// TwinCAT 3 PLC project IBF_Utilities
// Title: IBF_Utilities
// Company: Industrial Brains B.V.
// ProjectVersion: 0.0.0.0
// Description: The utilities library contains all basic utilities needed like system variables, messages, parameters etc.
// ProgramVersion: 3.1.4023.0
// libraries:
//   Tc2_Standard, * (Beckhoff Automation GmbH)
//   Tc2_System, * (Beckhoff Automation GmbH)
//   Tc2_Utilities, * (Beckhoff Automation GmbH)
//   Tc3_EventLogger, * (Beckhoff Automation GmbH)
//   Tc3_Module, * (Beckhoff Automation GmbH)
// project tree:
//   Average/ FB_RollingAverageLREAL.TcPOU (not stored), FB_RollingAverageTime.TcPOU (not stored), F_AverageLREAL.TcPOU (not stored), F_AverageTime.TcPOU (not stored)
//   BaseFunctions/ FB_Base.TcPOU, FB_FunctionBase.TcPOU
//   Compare/Functions/ Between.TcPOU, Between360deg.TcPOU (not stored)
//   Conversion/ DegS_To_Rpm.TcPOU (not stored), DegS_To_Rpm_And_MMin.TcPOU, DT_To_Str.TcPOU, Grey_To_Bin.TcPOU, MMin_To_Rpm_And_DegS.TcPOU (not stored), Rpm_To_DegS.TcPOU
//   FaultsAndMessages/DataTypes/ E_FaultTypes.TcTLEO, E_ResetState.TcDUT, UDT_Fault.TcDUT, UDT_FaultLogItem.TcDUT, UDT_Identity.TcDUT
//   FaultsAndMessages/Functions/ FB_FaultHandler.TcPOU
//   General/DataTypes/ E_ComponentTypes.TcTLEO, E_Locations.TcTLEO, Udt_TimerBandwith.TcDUT
//   GVLs/ DataManager.TcGVL, GVL_FixedValues.TcGVL, GVL_Parameters.TcGVL, GVL_Utilities.TcGVL, PAR_Utilities.TcGVL, Sys_Variables.TcGVL
//   Logger/DataTypes/ UDT_LogHandlerConfig.TcDUT, UDT_LogItem.TcDUT, E_LogLevel.TcDUT
//   Logger/Functions/ FB_Logger.TcPOU
//   Logger/Functions/LogHandlers/DataTypes/ E_LogToDiskState.TcDUT
//   Logger/Functions/LogHandlers/ FB_LogHandlerBase.TcPOU, FB_LogHandler_PersistentArray.TcPOU, FB_LogHandler_ADSLOG.TcPOU, FB_LogHandler_TxtFile.TcPOU
//   MovePathCalculations/ fAccDecCalc.TcPOU (not stored)
//   Parameter/DataTypes/ E_ParameterHandlerState.TcDUT, Udt_Parameter.TcDUT, Udt_ParameterId.TcDUT
//   Parameter/Functions/ FB_ParameterFileHandler.TcPOU, FB_ParameterHandler.TcPOU, F_ParToCsvLine.TcPOU (not stored)
//   PathFunctions/ F_FBNameFromPath.TcPOU (not stored), F_GetLevelFromPath.TcPOU (not stored)
//   / PlcTask.TcTTO
//   Positions/FunctionBlocks/ FB_PositionTrigger.TcPOU (not stored), FB_PositionTrigger_Old.TcPOU (not stored)
//   Positions/Functions/ F_AccDecDistanceFromTime.TcPOU (not stored), F_AccDecDistanceFromVelo.TcPOU (not stored), F_PosCheck.TcPOU, F_TopVelocityFromTime.TcPOU (not stored), F_TriggerPosOffset.TcPOU (not stored)
//   StateMachine/ FB_PauseableStateMachine.TcPOU, FB_StateMachine.TcPOU
//   StepFunctions/ FB_CycleTrigger.TcPOU (not stored), FB_Step.TcPOU
//   System/Functions/DataManagement/ FB_PersistentDataManager.TcPOU
//   System/Functions/ Fb_SystemVariables.TcPOU
//   _TESTS/ FB_Base_Test.TcPOU, PRG_TEST_CONVERSION.TcPOU, PRG_TEST_FB_BASE.TcPOU, PRG_TEST_FB_FAULTHANDLER.TcPOU, PRG_TEST_FB_LOGGER.TcPOU, PRG_TEST_FB_PARAMETERHANDLER.TcPOU, PRG_TEST_FB_PARFILEHANDLER.TcPOU, PRG_TEST_FB_STATEMACHINE.TcPOU, PRG_TEST_FB_PAUSEABLESTATEMACHINE.TcPOU, PRG_TEST_GLOBAL.TcPOU
// real-time tasks:
//   TASK PlcTask: cycle T#10ms, priority 20, ADS port 350

CONFIGURATION IBF_Utilities
    RESOURCE PLC ON TwinCAT3
        TASK PlcTask(INTERVAL := T#10ms, PRIORITY := 20);
        PROGRAM PRG_TEST_GLOBAL WITH PlcTask : PRG_TEST_GLOBAL;
        PROGRAM PRG_TEST_FB_BASE WITH PlcTask : PRG_TEST_FB_BASE;
        PROGRAM PRG_TEST_FB_FAULTHANDLER WITH PlcTask : PRG_TEST_FB_FAULTHANDLER;
        PROGRAM PRG_TEST_FB_PARAMETERHANDLER WITH PlcTask : PRG_TEST_FB_PARAMETERHANDLER;
        PROGRAM PRG_TEST_FB_PARFILEHANDLER WITH PlcTask : PRG_TEST_FB_PARFILEHANDLER;
        PROGRAM PRG_TEST_FB_STATEMACHINE WITH PlcTask : PRG_TEST_FB_STATEMACHINE;
        PROGRAM PRG_TEST_FB_PAUSEABLESTATEMACHINE WITH PlcTask : PRG_TEST_FB_PAUSEABLESTATEMACHINE;
        PROGRAM PRG_TEST_CONVERSION WITH PlcTask : PRG_TEST_CONVERSION;
        PROGRAM PRG_TEST_FB_LOGGER WITH PlcTask : PRG_TEST_FB_LOGGER;
    END_RESOURCE
END_CONFIGURATION

// ---- FaultsAndMessages/DataTypes/E_FaultTypes.TcTLEO
{attribute 'qualified_only'}
{attribute 'to_string'}
TYPE E_FaultTypes : // Fault types, sorted by severity
(
	OM, // Operator message
	OW, // Operator warning
	MC, // Missing condition
	CF, // Cycle Fault
	FF, // Fatal fault
	_ENUM_SIZE // Always the last item in the enumerator
) UINT;
END_TYPE

// ---- FaultsAndMessages/DataTypes/E_ResetState.TcDUT
{attribute 'qualified_only'}
{attribute 'strict'}
TYPE E_ResetState :
(
	Idle,
	ResetFaultTypes,
	WaitForFaults,
	Done
);
END_TYPE

// ---- FaultsAndMessages/DataTypes/UDT_Fault.TcDUT
TYPE UDT_Fault :
STRUCT
	Active 			: BOOL := FALSE;
	FaultType 		: E_FaultTypes;
	Description 	: STRING;
END_STRUCT
END_TYPE

// ---- FaultsAndMessages/DataTypes/UDT_FaultLogItem.TcDUT
TYPE UDT_FaultLogItem :
STRUCT
	bEmpty			: BOOL := TRUE; // This log item is empty (does not contain a fault)
	stFault 		: UDT_Fault;
	Id				: STRING; // Fault ID used for reporting and checking duplicates (not an unique value unless description matches as well)
	StartTime		: DATE_AND_TIME; // Time the fault became active
	EndTime			: DATE_AND_TIME; // Time the fault stopped being active
	nInactiveCycles	: UINT; // The number of PLC cycles the fault hasn't been active 
END_STRUCT
END_TYPE

// ---- FaultsAndMessages/DataTypes/UDT_Identity.TcDUT
TYPE UDT_Identity : // The identity is used for logging and fault handling
STRUCT
	nId				: UINT;
	nParentId		: UDINT; // Id of higher level object if aplicable (0 = no parent)
	nLocationId		: UDINT; // Unique Id calculated from Id and ParentId, used for parameter numbers, and as the parent ID for children
	eComponentType	: E_ComponentTypes;
	sName			: STRING[50];
END_STRUCT
END_TYPE

// ---- General/DataTypes/E_ComponentTypes.TcTLEO
{attribute 'qualified_only'}
{attribute 'strict'}
{attribute 'to_string'}
TYPE E_ComponentTypes :
(
	// No entry
		NA			:= 0,
	// Actuators 
		Cylinder 	:= 10,
		Axis		:= 11,
		Heaters		:= 12,
	// Buttons 
		EstopButton	:= 20,
		EstopBumper	:= 21,	
		Pushbutton 	:= 22,
		Switch		:= 23,
	// I/O
		SafeIO		:= 30,
		Rio_Box		:= 31,
		Rio_Slot	:= 32,
		Encoder		:= 33,
		DiInput		:= 34,
		AnInput		:= 35,
		DiOutput	:= 36,
		AnOutput	:= 37,
	// Drive
		ServoDrive 	:= 40,
	// Operation
		HMI			:= 50,
		RemoteOS	:= 51,
		RemoteDB	:= 52,
	// Assemblies
		Assembly 	:= 60,
		SubAssembly	:= 61,
	// functions
		MainProgram		:= 100,
		StepProgram		:= 101,
		FunctionBlock	:= 102 
)UDINT;
END_TYPE

// ---- General/DataTypes/E_Locations.TcTLEO
{attribute 'qualified_only'}
{attribute 'strict'}
TYPE E_Locations :
(
	MainPLC,
	MainPower_230V, 
	MainPower_24V, 
	MainAirSupply,
	MainScreen,
	MainIO,
	RemoteIO
);
END_TYPE

// ---- General/DataTypes/Udt_TimerBandwith.TcDUT
TYPE Udt_TimerBandwith :
STRUCT
	Minimal	:LREAL;// Timer values, Minimum time
	Nominal	:LREAL;// timer values, nominal time
	Maximum	:LREAL;// Timer values, Maximum time
END_STRUCT
END_TYPE

// ---- Logger/DataTypes/UDT_LogHandlerConfig.TcDUT
TYPE UDT_LogHandlerConfig :
STRUCT
	pLogHandler 		: POINTER TO FB_LogHandlerBase := 0;
	eMinimumLogLevel 	: E_LogLevel := E_LogLevel.TRACE;
END_STRUCT
END_TYPE

// ---- Logger/DataTypes/UDT_LogItem.TcDUT
TYPE UDT_LogItem :
STRUCT
	eLevel 		: E_LogLevel;
	stTimestamp : TIMESTRUCT;
	sMsg 		: STRING[255-2]; // Keep 2 bytes room for CRLF line ending
END_STRUCT
END_TYPE

// ---- Logger/DataTypes/E_LogLevel.TcDUT
{attribute 'qualified_only'}
{attribute 'strict'}
{attribute 'to_string'}
TYPE E_LogLevel : // Log levels, for more info see logger methods DEBUG, INFO, etc
(
	TRACE,
	DEBUG,
	INFO,
	WARN,
	ERROR,
	FATAL
) USINT;
END_TYPE

// ---- Logger/Functions/LogHandlers/DataTypes/E_LogToDiskState.TcDUT
{attribute 'qualified_only'}
{attribute 'strict'}
TYPE E_LogToDiskState : // LogToDisk state
(
	InitializeFBs,
	WaitForCommand,
	OpenOrCreateFile,
	CheckFileSize,
	WriteLogItemPrefix,
	WriteLogItemMessage,
	CloseFile,
	FindObsoleteFiles,
	DeleteFile,
	Error
) UDINT;
END_TYPE

// ---- Parameter/DataTypes/E_ParameterHandlerState.TcDUT
{attribute 'qualified_only'}
{attribute 'strict'}
TYPE E_ParameterHandlerState : // Parameter file handler state
(
	InitializeFBs,
	WaitForCommand,
	OpenExistingFile,
	CreateFile,
	WriteRecord,
	WriteRecordBusy,
	ReadRecord,
	ParseRecord,
	CloseFile,
	Error
);
END_TYPE

// ---- Parameter/DataTypes/Udt_Parameter.TcDUT
TYPE Udt_Parameter :
STRUCT PERSISTENT
	nNumber					: UDINT	 	:= 0						; // [Column 0]Parameter data, parameter number
	sName					: STRING	:= 'No parameter' 			; // [Column 1]Parameter data, Parameter name
	sType					: STRING	:= 'PPar'					; // [Column 2]Parameter data, Type of parameter [Mpar, Cpar, Opar, Ppar]
	sDiscription			: STRING	:= 'No parameter selected'	; // [Column 3]Parameter data, Parmater discription
	fFactory				: LREAL		:= 0						; // [Column 4]Parameter data, Factory standard value
	fMaximum				: LREAL		:= 0						; // [Column 5]Parameter data, Maximum parameter value
	fMinimum				: LREAL		:= 0						; // [Column 6]Parameter data, Minimum parameter value
	sUnit					: STRING	:= 'na'						; // [Column 7]Parameter data, Unit of measurement
	fValue					: LREAL		:= 0						; // [Column 8]Parameter data, Current (active) parameter value
	fSaved					: LREAL		:= 0						; // Parameter data, Saved value or standard setpoint
	fPrepared				: LREAL 	:= 0						; // Parameter data, Prepared value from teach function 
	bTeachable				: BOOL		:= FALSE					; // Teach command for devices 
	bAccepted				: BOOL 		:= FALSE 					; // Parameter value has been accepted
	bLoadedFromPersistent 	: BOOL 									; // The variable has been loaded for persistent memory, Note: No init value.
END_STRUCT
END_TYPE

// ---- Parameter/DataTypes/Udt_ParameterId.TcDUT
TYPE Udt_ParameterId :
STRUCT
	nNumber		: UDINT := 0 	; // parameter number
	sName		: STRING[50] := 'NA' ; // parameter name
	sType		: STRING[4]	:= 'Ppar'	; // parameter type 
	pParameter	: POINTER TO Udt_Parameter ; // pointer to parameter
END_STRUCT
END_TYPE

// ---- GVLs/DataManager.TcGVL
{attribute 'qualified_only'}
VAR_GLOBAL
	FbPersistentManager : FB_PersistentDataManager ;
END_VAR

// ---- GVLs/GVL_FixedValues.TcGVL
{attribute 'qualified_only'}
VAR_GLOBAL CONSTANT
	nINTMAXVALUE	: INT := 32767 		; // Integer maximum value 32767
	nINTMINVALUE	: INT := -32767		; // intiger minimum value -32767
	nDINTMAXVALUE	: DINT:= 2147483647 ; // Double integer maximum value 2,147,483,647
	nDINTMINVALUE	: DINT:= -2147483647; // Double integer minimum value -2,147,483,647
END_VAR

// ---- GVLs/GVL_Parameters.TcGVL
{attribute 'qualified_only'}
VAR_GLOBAL
	fbParameterHandler		: FB_ParameterFileHandler ; // Default parameter handler for visualisation and file handling
	sPARLIST_FILE			: T_MaxString 		:= 'D:\Parameters\ParameterList.csv';(* CSV destination file path and name *)
	sPARLOG_FILE			: T_MaxString 		:= 'D:\Parameters\ParameterLog.csv';(* CSV destination file path and name *)
END_VAR
VAR_GLOBAL CONSTANT
	MAX_PARAMETERS 			: UINT := 1000	;
	PAR_COLUMNS 			: UDINT := 8	;
	MAX_CSV_FIELD_LENGTH	: UDINT := 100	;
	sNetId					: T_AmsNetID		:= '' ;
END_VAR

// ---- GVLs/GVL_Utilities.TcGVL
{attribute 'qualified_only'}
VAR_GLOBAL
	fbFaultHandler : FB_FaultHandler; // The one and only faulthandler (a singleton)
END_VAR
VAR_GLOBAL CONSTANT
	// Not a PAR_Utility, because this constant is used by a HMI list (which is not compatible with configurable constant values)
	RETAINABLE_LOG_HISTORY_SIZE : UINT := 100;
END_VAR

// ---- GVLs/PAR_Utilities.TcGVL
{attribute 'qualified_only'}
// Contains library parameters
VAR_GLOBAL CONSTANT
	MAX_FAULTS_IN_LOG : UINT := 16; // Max number of faults in the FaultHandler log (should match with the size of the HMI's logview table)
END_VAR

// ---- GVLs/Sys_Variables.TcGVL
(* System variables *)
{attribute 'qualified_only'}
VAR_GLOBAL
// SystemFuntion
	fbSystemVariables : Fb_SystemVariables ;
	AlwaysOn		:BOOL 			;// System variable, Always on bit
	AlwaysOff		:BOOL 			;// System variable, Always off bit
	BlinkFast		:BOOL 			;// System variable, Blink fast bit 1sec 
	BlinkSlow		:BOOL 			;// System variable, Blink slow bit 2 sec
	Pulse1Sec		:BOOL 			;// System variable, Pulse 1 cycle every second
	Pulse100ms		:BOOL 			;// System variable, pulse 1 cycle every 100 ms
	SystemTime		:DATE_AND_TIME	; // System variable, Windows system time as DATE_AND_TIME
	SystemTime_TS	:TIMESTRUCT		; // System variable, Windows system time as TIMESTRUCT
	TimeZoneId		:E_TimeZoneID 	; // System variable, time zone Id 
	HeartBeat		:BOOL 			;// System Variable, Main system heartbeat 0.5 sec on 0.5 sec off
END_VAR

// ---- _TESTS/PRG_TEST_GLOBAL.TcPOU
PROGRAM INTERNAL PRG_TEST_GLOBAL // A place to call global function blocks (singletons) that can be used by all tests

Sys_Variables.fbSystemVariables();
GVL_Utilities.fbFaultHandler();

END_PROGRAM

// ---- _TESTS/PRG_TEST_FB_BASE.TcPOU
PROGRAM INTERNAL PRG_TEST_FB_BASE
VAR
	bEnableTests : BOOL;
	fbBase : FB_Base_Test;
END_VAR

IF bEnableTests THEN
	fbBase.Init(1, 2, E_ComponentTypes.MainProgram);
	fbBase();
END_IF

END_PROGRAM

// ---- _TESTS/FB_Base_Test.TcPOU
FUNCTION_BLOCK INTERNAL FB_Base_Test EXTENDS FB_Base

SUPER^();

METHOD PUBLIC Init : BOOL
VAR_INPUT
	nId				: UINT ; // Identification number of object
	nParentId		: UINT ; // Id of higher level if applicable (0 = no parent)
	eComponentType	: E_ComponentTypes ; // Component or function type
END_VAR
// Every FB_Base instance is expected to have an Init method that calls ExecIdentifyDevice. 
// This Init method will have at least the nId and nParentId inputs.
// The eComponentType input is optional (can be hardcoded in the Init method, for example see FB_Step).
// It might also have additional inputs (changing the method signature) therefore it is not declared in FB_Base.
ExecIdentifyDevice(nId,	nParentId,	eComponentType);
END_METHOD

END_FUNCTION_BLOCK

// ---- BaseFunctions/FB_Base.TcPOU
{attribute 'reflection'}
FUNCTION_BLOCK PUBLIC ABSTRACT FB_Base
VAR_INPUT
	bEnable			: BOOL 		:= TRUE 	; // Module enable signal reference Default := TRUE (when using system library := GVL_Main.stModules[nModuleId].bEnabled)
	refFbParHandler	: REFERENCE TO FB_ParameterFileHandler := GVL_Parameters.fbParameterHandler	; // reference to parameter handler
	bCmdPause 		: BOOL 		:= FALSE	; // Command Pause functions		
END_VAR
VAR_OUTPUT
	stIdentity 		: UDT_Identity;
	bInitOk			: BOOL 			:= FALSE 	; // function is initialized
	bBusy 			: BOOL 			:= FALSE 	; // device is busy
	bReady			: BOOL 			:= FALSE 	; // device is ready for new command 
	bErrorActive	: BOOL			:= FALSE	; // device Error active 
END_VAR
VAR
	stFault			: UDT_Fault		; // Fault data from device

	// Function path 
	{attribute 'instance-path'} 
    {attribute 'noinit'}
	sPath			: STRING	; // Path name of function (used for manual reference)
END_VAR

GVL_Utilities.fbFaultHandler.CmdAddFault(
	stFault := stFault,
	stIdentity := stIdentity
);

METHOD PUBLIC CmdReset : BOOL
VAR_INPUT
END_VAR
bErrorActive := FALSE ;

CmdReset := TRUE ;
END_METHOD

METHOD PROTECTED ExecIdentifyDevice : BOOL
VAR_INPUT
	nId				: UINT; // Identification number of object (between 0 and 99)
	nParentId		: UDINT; // Id of higher level If aplicable (0 = no parent)
	eComponentType	: E_ComponentTypes; // Component or function type
END_VAR
stIdentity.nId := nId;
stIdentity.nParentId := nParentId;
stIdentity.eComponentType := eComponentType;
stIdentity.sName := F_FBNameFromPath(sPath := sPath);
stIdentity.nLocationId := stIdentity.nParentId * 10000 + stIdentity.nId * 100;

ExecIdentifyDevice := (stIdentity.sName <> '') AND (stIdentity.nId < 100);
END_METHOD

END_FUNCTION_BLOCK

// ---- Parameter/Functions/FB_ParameterFileHandler.TcPOU
FUNCTION_BLOCK FB_ParameterFileHandler EXTENDS FB_ParameterHandler
VAR CONSTANT
	sCSVFileHeader 	: STRING := 'NUMBER;NAME;TYPE;DESCRIPTION;FACTORY;MAXIMUM;MINIMUM;UNIT;VALUE$L';
	CSV_FIELDS 		: UINT := 9;
END_VAR
VAR_OUTPUT
	bFault : BOOL;
	sFaultDescription : STRING;
END_VAR
VAR
	// States
	eState 		: E_ParameterHandlerState := E_ParameterHandlerState.InitializeFBs;
	
	// Command helpers
	bDone 		: BOOL;
	bCmdInit 	: BOOL;
	bCmdSavePar : BOOL;
	
	// File function blocks (asynchronous)
	fbFileOpen	: FB_FileOpen; // https://infosys.beckhoff.com/content/1033/tcplclib_tc2_system/30977547.html
	fbFileWrite	: FB_FileWrite; // https://infosys.beckhoff.com/content/1033/tcplclib_tc2_system/30986763.html
	fbFileClose	: FB_FileClose; // https://infosys.beckhoff.com/content/1033/tcplclib_tc2_system/30972939.html
	fbFileGets	: FB_FileGets; // https://infosys.beckhoff.com/content/1033/tcplclib_tc2_system/30976011.html

	// CSV handling
	sCsvRecord : T_MaxString := ''; // String buffer (single CSV text line)
	bHeaderRead : BOOL; // TRUE once the CSV header line has been read
	fbCsvMemBufReader : FB_CSVMemBufferReader; // https://infosys.beckhoff.com/content/1033/tcplclib_tc2_utilities/34977931.html
	fbCsvMemBufWriter : FB_CSVMemBufferWriter; // https://infosys.beckhoff.com/content/1033/tcplclib_tc2_utilities/34979467.html

	// Miscelleanous
	nIdxPar  : UINT; // Parameter array iterator
END_VAR

ExecStateMachine();

METHOD PUBLIC CmdSavePar : BOOL
IF NOT bCmdSavePar THEN
	bDone := FALSE;
	bCmdSavePar := TRUE;
ELSIF bDone THEN
	bCmdSavePar := FALSE;
END_IF	

CmdSavePar := bDone;
END_METHOD

METHOD PRIVATE ExecStateMachine : BOOL
VAR
	i 					: UINT; // Iterator
	pParameter 			: POINTER TO Udt_Parameter; // Temporary pointer to parameter
	sParameterFromFile 	: Udt_Parameter; // Parameter retrieved from file
	sCSVField 			: T_MaxString; // Single CSV field value (record field)
	bMatch 				: BOOL;
END_VAR
// Parameter file handler state machine
CASE eState OF
	E_ParameterHandlerState.InitializeFBs:
		// Initialize function blocks
		fbFileOpen(
			bExecute := FALSE,
			ePath := PATH_GENERIC,
		);
		fbFileWrite(
			bExecute := FALSE,
			pWriteBuff := ADR(sCsvRecord)
		);
		fbFileClose(bExecute := FALSE);
		fbFileGets(bExecute := FALSE);

		fbCsvMemBufWriter.pBuffer := ADR(sCsvRecord);
		fbCsvMemBufReader.pBuffer := ADR(sCsvRecord);
		fbCsvMemBufWriter.cbBuffer := SIZEOF(sCsvRecord) - 1;
		fbCsvMemBufReader.cbBuffer := SIZEOF(sCsvRecord);
	
		eState := E_ParameterHandlerState.WaitForCommand;

	E_ParameterHandlerState.WaitForCommand:
		sFaultDescription := '';
		IF bCmdInit THEN
			eState := E_ParameterHandlerState.OpenExistingFile;
		ELSIF bCmdSavePar THEN
			eState := E_ParameterHandlerState.CreateFile;
		END_IF	

	E_ParameterHandlerState.OpenExistingFile:
		fbFileOpen(
			bExecute := TRUE,	
			sPathName := GVL_Parameters.sPARLIST_FILE,
			nMode := FOPEN_MODEREAD OR FOPEN_MODETEXT, // Open file in read only text mode
		);

		IF (NOT fbFileOpen.bBusy) THEN
			fbFileOpen(bExecute := FALSE);

			IF fbFileOpen.bError THEN
				// Check error codes
				IF (fbFileOpen.nErrId = 16#70C) THEN
					// File not found
					eState := E_ParameterHandlerState.CreateFile;
				ELSE
					sFaultDescription := 'Unable to open file';
					eState := E_ParameterHandlerState.Error;
				END_IF
			ELSE
				nIdxPar := 0;
				bHeaderRead := FALSE;
				eState := E_ParameterHandlerState.ReadRecord;
			END_IF
		END_IF

	E_ParameterHandlerState.CreateFile:
		fbFileOpen(
			bExecute := TRUE,	
			sPathName := GVL_Parameters.sPARLIST_FILE,
			nMode := FOPEN_MODEWRITE OR FOPEN_MODETEXT, // Open file in read/write text mode
		);

		IF (NOT fbFileOpen.bBusy) THEN
			fbFileOpen(bExecute := FALSE);

			IF fbFileOpen.bError THEN
				sFaultDescription := 'Unable to create file';
				eState := E_ParameterHandlerState.Error;
			ELSE		
				fbFileWrite.hFile := fbFileOpen.hFile;
				nIdxPar := 0;
				eState := E_ParameterHandlerState.WriteRecord;
			END_IF
		END_IF
		
	E_ParameterHandlerState.WriteRecord:
		// Code based on Beckhoff example: https://infosys.beckhoff.com/content/1033/tcplclib_tc2_utilities/34979467.html
		sCsvRecord := '';
		fbCsvMemBufWriter.eCmd := eEnumCmd_First; // Write first field value

		IF (nIdxPar > nNumberOfParameters) THEN
			// Done (all parameters were added)
			eState := E_ParameterHandlerState.CloseFile;
		ELSIF (nIdxPar = 0) THEN
			// First line: write the CSV header
			sCsvRecord := sCSVFileHeader;
			eState := E_ParameterHandlerState.WriteRecordBusy;
		ELSE
			// Add the next parameter
			pParameter := arParameters[nIdxPar].pParameter;
			IF (pParameter = 0) THEN
				sFaultDescription := 'Unexpected null pointer';
				eState := E_ParameterHandlerState.Error;
			ELSE
				// Save current actual value for later restore
				pParameter^.fSaved := pParameter^.fValue;
				// Create CSV record
				FOR i := 1 TO CSV_FIELDS DO 
					CASE i OF
						1: sCSVField := UDINT_TO_STRING(pParameter^.nNumber);
						2: sCSVField := pParameter^.sName;
						3: sCSVField := pParameter^.sType;
						4: sCSVField := pParameter^.sDiscription;
						5: sCSVField := LREAL_TO_STRING(pParameter^.fFactory);
						6: sCSVField := LREAL_TO_STRING(pParameter^.fMaximum);
						7: sCSVField := LREAL_TO_STRING(pParameter^.fMinimum);
						8: sCSVField := pParameter^.sUnit;
						9: sCSVField := LREAL_TO_STRING(pParameter^.fValue);
					END_CASE
					sCSVField := STRING_TO_CSVFIELD(sCSVField, FALSE);
					
					// Add new field to the record buffer
					fbCsvMemBufWriter(
						putValue := sCSVField,
						bCRLF := (i = CSV_FIELDS) // Write CRLF after the last field value 
					);
					IF fbCsvMemBufWriter.bOk THEN
						fbCsvMemBufWriter.eCmd := eEnumCmd_Next;
					ELSE // Error
						sFaultDescription := 'Unable to store fields in CSV buffer';
						eState := E_ParameterHandlerState.Error;
						RETURN;
					END_IF
	
				END_FOR

				eState := E_ParameterHandlerState.WriteRecordBusy;
			END_IF;
		END_IF;

	E_ParameterHandlerState.WriteRecordBusy:
		fbFileWrite(bExecute := TRUE, cbWriteLen := INT_TO_UDINT(LEN(sCsvRecord)));
		IF (NOT fbFileWrite.bBusy) THEN
			fbFileWrite(bExecute := FALSE);
			IF fbFileWrite.bError THEN
				sFaultDescription := 'Unable to write record to file';
				eState := E_ParameterHandlerState.Error;
			ELSE		
				nIdxPar := nIdxPar + 1;	 
				eState := E_ParameterHandlerState.WriteRecord;
			END_IF
		END_IF
		
	E_ParameterHandlerState.ReadRecord:
		fbFileGets(bExecute := TRUE, hFile := fbFileOpen.hFile);
		IF (NOT fbFileGets.bBusy) THEN
			sCsvRecord := fbFileGets.sLine;
			fbFileGets(bExecute := FALSE);
			IF fbFileGets.bError THEN
				sFaultDescription := 'Unable to read line from file';
				eState := E_ParameterHandlerState.Error;
			ELSIF fbFileGets.bEOF THEN
				// Finished reading the file
				eState := E_ParameterHandlerState.CloseFile;			
			ELSIF NOT bHeaderRead THEN 
				// Skip first line (header)
				bHeaderRead := TRUE;
			ELSE
				eState := E_ParameterHandlerState.ParseRecord;
			END_IF
		END_IF

	E_ParameterHandlerState.ParseRecord:
		fbCsvMemBufReader.eCmd := eEnumCmd_First; // Read first field value

		FOR i := 1 TO CSV_FIELDS DO 
			// Read field from the record buffer
			fbCsvMemBufReader(getValue => sCSVField);
			IF fbCsvMemBufReader.bOk THEN
				sCSVField := CSVFIELD_TO_STRING(sCSVField, FALSE);
				CASE i OF
					1: sParameterFromFile.nNumber := STRING_TO_UDINT(sCSVField);
					2: sParameterFromFile.sName := sCSVField;
					3: sParameterFromFile.sType := sCSVField;
					4: sParameterFromFile.sDiscription := sCSVField;
					5: sParameterFromFile.fFactory := STRING_TO_LREAL(sCSVField);
					6: sParameterFromFile.fMaximum := STRING_TO_LREAL(sCSVField);
					7: sParameterFromFile.fMinimum := STRING_TO_LREAL(sCSVField);
					8: sParameterFromFile.sUnit := sCSVField;
					9: sParameterFromFile.fValue := STRING_TO_LREAL(sCSVField);
				END_CASE
				
				fbCsvMemBufReader.eCmd := eEnumCmd_Next;
			ELSE // Error
				sFaultDescription := 'Unable to parse all CSV fields';
				eState := E_ParameterHandlerState.Error;
				RETURN;
			END_IF
		END_FOR
			
		// Done reading parameter from file. Search for parameter in the PLC parameter array, and copy values.
		FOR i := 1 TO nNumberOfParameters DO
			pParameter := arParameters[i].pParameter;
			IF (pParameter = 0) THEN
				// Unexpected null pointer
				EXIT;
			ELSIF (sParameterFromFile.nNumber = pParameter^.nNumber) THEN
				bMatch := TRUE;
				pParameter^.sName := sParameterFromFile.sName;
				pParameter^.sType := sParameterFromFile.sType;
				pParameter^.sDiscription := sParameterFromFile.sDiscription;
				pParameter^.fFactory := sParameterFromFile.fFactory;
				pParameter^.fMaximum := sParameterFromFile.fMaximum;
				pParameter^.fMinimum := sParameterFromFile.fMinimum;
				pParameter^.sUnit := sParameterFromFile.sUnit;
				pParameter^.fValue := sParameterFromFile.fValue;
				EXIT;
			END_IF
		END_FOR

		IF bMatch THEN
			// Finished, move to the next record		
			eState := E_ParameterHandlerState.ReadRecord;
		ELSE
			sFaultDescription := 'Parameter in CSV file not found in PLC';
			eState := E_ParameterHandlerState.Error;
		END_IF
	
	E_ParameterHandlerState.CloseFile:
		fbFileClose(bExecute := TRUE, hFile := fbFileOpen.hFile);
		IF (NOT fbFileClose.bBusy) THEN
			fbFileClose(bExecute := FALSE);
			IF fbFileClose.bError THEN
				sFaultDescription := 'Unable to close file'; 
				eState := E_ParameterHandlerState.Error;
			ELSE
				bDone := TRUE;
				eState := E_ParameterHandlerState.WaitForCommand;
			END_IF
		END_IF
	
	E_ParameterHandlerState.Error:
		IF (sFaultDescription = '') THEN
			sFaultDescription := 'Unknown error';
		END_IF

END_CASE

bFault := (eState = E_ParameterHandlerState.Error);
END_METHOD

METHOD PUBLIC Init : BOOL
IF NOT bCmdInit THEN
	bDone := FALSE;
	bCmdInit := TRUE;
ELSIF bDone THEN
	bCmdInit := FALSE;
END_IF	

Init := bDone;
END_METHOD

END_FUNCTION_BLOCK

// ---- Parameter/Functions/FB_ParameterHandler.TcPOU
FUNCTION_BLOCK PUBLIC FB_ParameterHandler
VAR_OUTPUT
	arParameters		: ARRAY [1..GVL_Parameters.MAX_PARAMETERS] OF Udt_ParameterId := [stDummyParId]; 
END_VAR
VAR
	nLookupIndex		: UINT := 1;
	nNumberOfParameters : UINT := 1;
	// parameter change commands
	bCmdLoadfactory		: BOOL 	:= FALSE; // Load factory value into prepared value 
	bCmdLoadFromPrevious: BOOL 	:= FALSE; // Load from saved previous value into prepared value
	bCmdTeach			: BOOL 	:= FALSE; // Start teaching function for selected parameter
	bCmdAcceptTeach		: BOOL 	:= FALSE ; // Accept the teach value
	// Dummy parameter when no parameters are added yet
	stDummyParId		: Udt_ParameterId ;
	// Memory 
	fValueOld			: LREAL	:= 0 ; // previous value
END_VAR

// call parameter change function 
ExecChangeParValues();

METHOD PUBLIC CmdAddParameter : BOOL
VAR_IN_OUT
	refParameter : Udt_Parameter ; // Parameter to add
END_VAR
VAR
	i 			: UINT ;
	j			: UINT ;
	stTempPar	: Udt_ParameterId ;
	bParFound	: BOOL 	:= FALSE ;
END_VAR
//Single loop to get the number of parameters and check if that parameter has already been added  
FOR i := 1 TO GVL_Parameters.MAX_PARAMETERS DO
	//Check if it's a valid reference
	IF (arParameters[i].pParameter = 0) THEN
		//No, we have reached the end of the list
		//The current index - 1 is the ammount of parameters
		nNumberOfParameters := i - 1;
		//Abort the FOR loop, we found the end.
		EXIT ;
	//It is a valid reference, valitate it is not already in the list  
	ELSIF arParameters[i].nNumber = refParameter.nNumber THEN
		//It is in the list, validate if the name matches 
		IF (arParameters[i].sName = refParameter.sName) THEN
			//Name and number match, assume it is the same parameter and just return that it is (already) added
			CmdAddParameter := TRUE;
			RETURN;
		ELSE
			//Number matches but not the name, this is a different parameter. Abort the add.
			CmdAddParameter := FALSE;
			RETURN;
		END_IF
	END_IF
END_FOR

//Ok, here we are shure it's a new parameter, try adding it to the array
nNumberOfParameters := nNumberOfParameters + 1; 
//Does it fit?
IF nNumberOfParameters <= GVL_Parameters.MAX_PARAMETERS THEN
	//It fits, store the data
	arParameters[nNumberOfParameters].nNumber		:= refParameter.nNumber 	;
	arParameters[nNumberOfParameters].sName			:= refParameter.sName	;
	arParameters[nNumberOfParameters].sType			:= refParameter.sType	;
	arParameters[nNumberOfParameters].pParameter 	:= ADR(refParameter)	;
	
	//Check if the add was sucessfull
	CmdAddParameter := arParameters[nNumberOfParameters].pParameter <> 0;
	
	//Give the command to (re)sort the parameter list
	ExecSortParameters();
ELSE
	//Does not fit, return FALSE
	CmdAddParameter := FALSE;	
END_IF
END_METHOD

METHOD ExecChangeParValues : BOOL
VAR
END_VAR
IF arParameters[nLookupIndex].pParameter <> 0 THEN 
	;
ELSE
	RETURN; 
END_IF

// Load values from default or saved
IF bCmdLoadfactory THEN 
	arParameters[nLookupIndex].pParameter^.fValue := arParameters[nLookupIndex].pParameter^.fFactory ;
	bCmdLoadfactory := FALSE ;
ELSIF bCmdLoadFromPrevious THEN
	arParameters[nLookupIndex].pParameter^.fValue := arParameters[nLookupIndex].pParameter^.fSaved ;
	bCmdLoadFromPrevious := FALSE ;
ELSIF bCmdAcceptTeach THEN 
	arParameters[nLookupIndex].pParameter^.fValue := arParameters[nLookupIndex].pParameter^.fPrepared ;
	bCmdAcceptTeach := FALSE ;
END_IF
END_METHOD

METHOD PRIVATE ExecSortParameters : BOOL
VAR_INPUT
END_VAR
VAR
	i 			: UDINT ;
	j			: UDINT ;
	stTempPar	: Udt_ParameterId ;
END_VAR
// (re)sort parameter list so it's order remains constant
FOR i := 2 TO nNumberOfParameters BY 1 DO
	FOR j := 1 TO nNumberOfParameters - 1 BY 1 DO
		IF (arParameters[j].nNumber > arParameters[j+1].nNumber)THEN
			stTempPar 			:= arParameters[j+1];
			arParameters[j+1]	:= arParameters[j];
			arParameters[j]		:= stTempPar ;
		END_IF
	END_FOR
END_FOR
END_METHOD

END_FUNCTION_BLOCK

// ---- _TESTS/PRG_TEST_FB_FAULTHANDLER.TcPOU
PROGRAM INTERNAL PRG_TEST_FB_FAULTHANDLER
VAR
	bEnableTests : BOOL;
	fbBase : FB_Base_Test;
	bCmdReset : BOOL;
	bCmdClearInactive : BOOL;
	stLogItem : UDT_FaultLogItem;
	bHead : BOOL;
	bNext : BOOL;
	bActive : BOOL;
	pFault : POINTER TO UDT_Fault; // Workaround to reach non-output variable fbBase.stFault
END_VAR

IF bEnableTests THEN
	fbBase();
	
	pFault := ADR(fbBase.stFault);
	pFault^.Active := bActive;
	
	IF bCmdReset THEN
		bCmdReset R= GVL_Utilities.fbFaultHandler.CmdReset();
	END_IF
	
	IF bCmdClearInactive THEN
		bCmdClearInactive R= GVL_Utilities.fbFaultHandler.CmdClearInactive();
	END_IF
	
	IF bHead THEN
		bHead := FALSE;
		stLogItem := GVL_Utilities.fbFaultHandler.Head;
	END_IF

	IF bNext THEN
		bNext := FALSE;
		stLogItem := GVL_Utilities.fbFaultHandler.Next;
	END_IF
END_IF

END_PROGRAM

// ---- _TESTS/PRG_TEST_FB_PARAMETERHANDLER.TcPOU
PROGRAM INTERNAL PRG_TEST_FB_PARAMETERHANDLER
VAR
	bEnableTests : BOOL;
	fbParameterHandler 	: FB_ParameterHandler;
	stParameterId		: Udt_ParameterId;
	stParameter 		: Udt_Parameter; // NOTE: Udt_Parameter is persistent
	bAddParameter 		: BOOL;
END_VAR

IF bEnableTests THEN
	fbParameterHandler();
	
	IF bAddParameter THEN
		bAddParameter := FALSE;
		fbParameterHandler.CmdAddParameter(stParameter);
	END_IF
END_IF

END_PROGRAM

// ---- _TESTS/PRG_TEST_FB_PARFILEHANDLER.TcPOU
PROGRAM INTERNAL PRG_TEST_FB_PARFILEHANDLER
VAR
	bEnableTests : BOOL;
	fbParFileHandler: FB_ParameterFileHandler;
	stParameter 	: Udt_Parameter; // NOTE: Udt_Parameter is persistent
	bAddParameter 	: BOOL;
	bInit			: BOOL;
	bCmdSavePar		: BOOL;
END_VAR

IF bEnableTests THEN
	fbParFileHandler();
	
	IF bAddParameter THEN
		bAddParameter := FALSE;
		fbParFileHandler.CmdAddParameter(stParameter);
	END_IF
	
	IF bInit THEN
		bInit R= fbParFileHandler.Init();
	END_IF
	
	IF bCmdSavePar THEN
		bCmdSavePar R= fbParFileHandler.CmdSavePar();
	END_IF
END_IF

END_PROGRAM

// ---- _TESTS/PRG_TEST_FB_STATEMACHINE.TcPOU
PROGRAM INTERNAL PRG_TEST_FB_STATEMACHINE
VAR
	bEnableTests : BOOL;
	nState : UDINT;
	fbStateMachine : FB_StateMachine;
	bStateChanged : BOOL; // A helper variable to detect bStateChanged output changes in FB_StateMachine
	nTimeInState : UDINT; // [msec] A helper variable to get the elapsed time as a number 
END_VAR

IF bEnableTests THEN
	fbStateMachine(nState := nState);
	bStateChanged S= fbStateMachine.bStateChanged;
	nTimeInState := TIME_TO_UDINT(fbStateMachine.tTimeInState);
END_IF

END_PROGRAM

// ---- StateMachine/FB_StateMachine.TcPOU
FUNCTION_BLOCK FB_StateMachine // A basic statemachine with some convenient outputs
VAR CONSTANT
	MAX_TIME : TIME := UDINT_TO_TIME(16#FFFFFFFF);
END_VAR
VAR_IN_OUT
	nState : UDINT;
END_VAR
VAR_OUTPUT
	tTimeInState : TIME;
	bStateChanged : BOOL;
END_VAR
VAR
	nStatePrev : UDINT;
	tonTimeInState : TON;
END_VAR

bStateChanged := (nStatePrev <> nState);
nStatePrev := nState;
tonTimeInState(IN := NOT bStateChanged, PT := MAX_TIME);
tTimeInState := tonTimeInState.ET;

END_FUNCTION_BLOCK

// ---- _TESTS/PRG_TEST_FB_PAUSEABLESTATEMACHINE.TcPOU
PROGRAM INTERNAL PRG_TEST_FB_PAUSEABLESTATEMACHINE
VAR CONSTANT
	PAUSE_STATE : UDINT := 100;
END_VAR
VAR
	bEnableTests : BOOL;

	nState : UDINT;
	fbStateMachine : FB_PauseableStateMachine;
	bDoSomething : BOOL;
END_VAR

IF bEnableTests THEN
	fbStateMachine(nState := nState, nPauseState := PAUSE_STATE);
	
	CASE nState OF
		0 : IF bDoSomething THEN
				nState := 1;
			END_IF
			
		PAUSE_STATE :
			IF bDoSomething THEN
				 fbStateMachine.Resume();
			END_IF
	END_CASE

	bDoSomething := FALSE;
END_IF

END_PROGRAM

// ---- StateMachine/FB_PauseableStateMachine.TcPOU
FUNCTION_BLOCK FB_PauseableStateMachine EXTENDS FB_StateMachine // An extension of FB_StateMachine that allows state pauses
VAR_INPUT
	nPauseState : UDINT; // The state to go to when paused
	bRequestPause : BOOL; // If TRUE, the state machine will go to nPauseState on the next state change
	bIgnorePause : BOOL; // If TRUE, the state machine will ignore a pause request. NOTE: This BOOL will be set to FALSE on a state change
END_VAR
VAR
	nResumeState : UDINT; // The state to go to when un-pausing (where the statemachine wanted to go, but wasn' allowed to) 
END_VAR

SUPER^(nState := nState);

IF bStateChanged THEN
	IF bRequestPause AND (NOT bIgnorePause) THEN
		nResumeState := nState;
		nState := nPauseState;
		nStatePrev := nState;
	END_IF
	bIgnorePause := FALSE;
END_IF

METHOD PUBLIC Resume
{warning disable C0371}
IF __ISVALIDREF(nState) THEN
	IF (NOT bRequestPause) THEN
		nState := nResumeState;
	END_IF
END_IF
{warning restore C0371}
END_METHOD

END_FUNCTION_BLOCK

// ---- _TESTS/PRG_TEST_CONVERSION.TcPOU
PROGRAM INTERNAL PRG_TEST_CONVERSION
VAR
 	bEnableTests : BOOL;

	in_dt : DATE_AND_TIME;
	out_str : STRING;
END_VAR

IF bEnableTests THEN
	out_str := Dt_To_Str(in_dt);
END_IF

END_PROGRAM

// ---- Conversion/DT_To_Str.TcPOU
FUNCTION DT_To_Str : STRING[19] // Takes a DATE_AND_TIME and converts it into a atring. If 0, an empty string is returned 
VAR_INPUT
	value : DATE_AND_TIME;
END_VAR
VAR
	str : STRING;
END_VAR

IF (DT_TO_DWORD(value) = 0) THEN
	DT_To_Str := '';
ELSE
	// Example input: 'DT#1998-02-13-14:20:00
	str := MID(DT_TO_STRING(value), 19, 4); // Cut off 'DT#'
	str := REPLACE(str, ' ', 1, 11); // Take out unnecessary '-'
	DT_To_Str :=  str;
END_IF

END_FUNCTION

// ---- _TESTS/PRG_TEST_FB_LOGGER.TcPOU
PROGRAM INTERNAL PRG_TEST_FB_LOGGER
VAR
	fbLogHandler_TxtFile :	FB_LogHandler_TxtFile(
									sLogFolder := 'D:\Temp\',
									sLogFilePrefix := 'AutomaticTestLog_',
									sLogFileExtension := 'txt',
									nMaxLogFileSize := 500,
									nMaxNumberOfLogFiles := 3
								);
	fbLogHandler_ADSLOG : FB_LogHandler_ADSLOG;
	fbLogger : FB_Logger;
	
	bRegisterLogHandlers : BOOL;
	bEnableTests : BOOL;
	bAddToLog : BOOL;
	eLogLevel : E_LogLevel;
	bStressTest : BOOL;
	nIdx : UDINT;
	sMsg : T_MaxString;
END_VAR

IF bEnableTests THEN
	IF bRegisterLogHandlers THEN
		fbLogger.RegisterLogHandler(fbLogHandler_ADSLOG, E_LogLevel.TRACE);
		fbLogger.RegisterLogHandler(fbLogHandler_TxtFile, E_LogLevel.TRACE);
	END_IF
	
	fbLogger.Run();
	
	IF bAddToLog THEN
		bAddToLog := FALSE;
		CASE eLogLevel OF
			E_LogLevel.TRACE:	fbLogger.TRACE(sMsg);
			E_LogLevel.DEBUG: 	fbLogger.DEBUG(sMsg);
			E_LogLevel.INFO: 	fbLogger.INFO(sMsg);
			E_LogLevel.WARN: 	fbLogger.WARN(sMsg);
			E_LogLevel.ERROR:	fbLogger.ERROR(sMsg);
			E_LogLevel.FATAL: 	fbLogger.FATAL(sMsg);
		END_CASE
	END_IF
	
	IF bStressTest THEN
		// Write an item to the log every PLC cycle, this should trigger a buffer overflow
		nIdx := nIdx + 1;
		sMsg := UDINT_TO_STRING(nIdx);
		fbLogger.TRACE(sMsg);
	END_IF
END_IF

END_PROGRAM

// ---- Logger/Functions/LogHandlers/FB_LogHandler_TxtFile.TcPOU
FUNCTION_BLOCK PUBLIC FB_LogHandler_TxtFile EXTENDS FB_LogHandlerBase // Regularly writes contents of the log to disk
// Once the log file reaches a set size, a new log file is created.
// If the max number of files is reached, the oldest file is discarded.
VAR CONSTANT
	MAX_ITEMS_IN_BUFFER : UDINT := 20; // Should be long enough to allow for worst case writes (where an old file has to be deleted and a new file created).  
END_VAR
VAR_OUTPUT
	bFault 				: BOOL; // An error occured while trying to add to log or write to disk
	sFaultDescription	: STRING[80]; // Detailed error information
	bLoggerInitialized  : BOOL; // True the first time the logger has ran through all states (ie., after succesfully writing the first log message and emptying the buffer)
	sCurrentLogFile		: T_MaxString; // The file which is currently used for logging (and can be viewed for instance by the HMI)
END_VAR
VAR
	// Properties set by FB_init
	sLogFolder 			: T_MaxString;
	sLogFilePrefix 		: T_MaxString;
	sLogFileExtension 	: T_MaxString;
	nMaxLogFileSize 	: ULINT; // [bytes] When this size is reached, a new log file is created 
	nMaxNumberOfLogFiles: UINT;

	// State machine
	fbStateMachine 	: FB_StateMachine;	
	eState 			: E_LogToDiskState := E_LogToDiskState.InitializeFBs;
	
	// Log item buffer
	stLogItemFromBuffer : UDT_LogItem; // Log item retrieved from the buffer	
	stLogItemToDisk		: UDT_LogItem; // Log item to be written to the log file
	cbBuffer 	: ARRAY[1..(MAX_ITEMS_IN_BUFFER * (SIZEOF(UDT_LogItem) + 4))] OF BYTE; // Note that the buffer size is larger than the number of items * item size, because 4 bytes are added to each item by FB_MemRingBuffer
	fbBuffer 	: FB_MemRingBuffer := (pBuffer:= ADR(cbBuffer), cbBuffer:= SIZEOF(cbBuffer));

	// File function blocks (asynchronous)
	fbFileOpen			: FB_FileOpen; // https://infosys.beckhoff.com/content/1033/tcplclib_tc2_system/30977547.html
	fbFilePuts			: FB_FilePuts; // https://infosys.beckhoff.com/content/1033/tcplclib_tc2_system/30979083.html
	fbFileClose			: FB_FileClose; // https://infosys.beckhoff.com/content/1033/tcplclib_tc2_system/30972939.html
	fbFileProperties	: FB_FileProperties; // https://infosys.beckhoff.com/content/1033/tcplclib_tc2_utilities/10047843595.html
    fbEnumFiles			: FB_EnumFindFileEntry; // https://infosys.beckhoff.com/content/1033/tcplclib_tc2_utilities/34982539.html
	fbFileDelete		: FB_FileDelete; // https://infosys.beckhoff.com/content/1033/tcplclib_tc2_system/30974475.html

	sPath: STRING; // Path to the current log file
	
	tOldestLogFile 	: ST_FindFileEntry; // Reference to the oldest log file in the log folder
	nFileCount		: UINT; // Number of log files found  
	
	fbFormatString : FB_FormatString; // https://infosys.beckhoff.com/content/1033/tcplclib_tc2_utilities/34990219.html
END_VAR
VAR_TEMP
	sTimestamp : T_MaxString;
	sLevel : T_MaxString;

	nFileSize : ULINT;
	
	stEmptyLogItem : UDT_LogItem;
END_VAR

fbStateMachine(nState := eState);

CASE eState OF
	E_LogToDiskState.InitializeFBs:
		// Initialize function blocks
		fbFileOpen(
			bExecute := FALSE,
			ePath := PATH_GENERIC,
		);
		fbFilePuts(bExecute := FALSE);
		fbFileClose(bExecute := FALSE);
		fbFileProperties(bExecute := FALSE);
		fbEnumFiles(bExecute := FALSE);
		fbFileDelete(
			bExecute := FALSE,
			ePath := PATH_GENERIC,
		);
		
		eState := E_LogToDiskState.WaitForCommand;

	E_LogToDiskState.WaitForCommand:
		IF (stLogItemFromBuffer.sMsg = '') THEN
			stLogItemFromBuffer := Pop();
		ELSE
			eState := E_LogToDiskState.OpenOrCreateFile;
		END_IF

	E_LogToDiskState.OpenOrCreateFile:
		IF fbStateMachine.bStateChanged THEN
			// Create a new file path if none was given (i.e., after reboot or when file size limit has been reached)
			IF (sPath = '') THEN
				sPath := CreatePath();
			END_IF  	
		END_IF
		fbFileOpen(
			bExecute := TRUE,	
			sPathName := sPath, 
			nMode := FOPEN_MODEAPPEND OR FOPEN_MODETEXT, // Open file in read/write text mode
		);
		IF (NOT fbFileOpen.bBusy) THEN
			fbFileOpen(bExecute := FALSE);
			IF fbFileOpen.bError THEN
				fbFormatString(sFormat := 'Unable to open file (error code 0x%X)', arg1 := F_UDINT(fbFileOpen.nErrId), sOut => sFaultDescription);
				eState := E_LogToDiskState.Error;
			ELSE
				sCurrentLogFile := sPath;
				eState := E_LogToDiskState.CheckFileSize;
			END_IF
		END_IF

	E_LogToDiskState.CheckFileSize:
		fbFileProperties(
			bExecute := TRUE,	
			sPathName := sPath 
		);
		IF (NOT fbFileProperties.bBusy) THEN
			fbFileProperties(bExecute := FALSE);
			IF fbFileProperties.bError THEN
				fbFormatString(sFormat := 'Unable to get file properties (error code 0x%X)', arg1 := F_UDINT(fbFileProperties.nErrId), sOut => sFaultDescription);
				eState := E_LogToDiskState.Error;
			ELSE
				// Check file size
				// ST_FindFileEntry info at https://infosys.beckhoff.com/content/1033/tcplclib_tc2_utilities/35363851.html
				nFileSize := ULARGE_TO_ULINT(fbFileProperties.stProperties.fileSize);
				IF (nFileSize >= nMaxLogFileSize) THEN
					// Create a final log item for this log file
					stLogItemToDisk.eLevel := E_LogLevel.DEBUG;
					fbFormatString(
						sFormat := 'File size exceeded (%u/%u bytes), creating new file.',
						arg1 := F_ULINT(nFileSize),
						arg2 := F_ULINT(nMaxLogFileSize),
						sOut => stLogItemToDisk.sMsg
					);
					stLogItemToDisk.stTimestamp := Sys_Variables.SystemTime_TS;
					sPath := ''; // Trigger new file creation
				ELSE
					stLogItemToDisk := stLogItemFromBuffer; // Set log item to be written to disk
					stLogItemFromBuffer := stEmptyLogItem; // Clear log item from buffer to trigger new item pop
				END_IF
				eState := E_LogToDiskState.WriteLogItemPrefix;
			END_IF
		END_IF
	
	E_LogToDiskState.WriteLogItemPrefix:
		IF fbStateMachine.bStateChanged THEN
			// Build a prefix string, e.g. '[2022-02-04 12:13:45.343] INFO; '

			// Suppress error "VAR_IN_OUT parameter 'in' needs variable with write access as input."	
			sLevel := TO_STRING(stLogItemToDisk.eLevel);
			sTimestamp := SYSTEMTIME_TO_STRING(stLogItemToDisk.stTimestamp);
 
			fbFormatString(
				sFormat := '[%s] %s: ',
				arg1 := F_STRING(sTimestamp),
				arg2 := F_STRING(sLevel),
				sOut => fbFilePuts.sLine
			);
		END_IF
		fbFilePuts(bExecute := TRUE, hFile := fbFileOpen.hFile);
		IF (NOT fbFilePuts.bBusy) THEN
			fbFilePuts(bExecute := FALSE);
			IF fbFilePuts.bError THEN
				fbFormatString(sFormat := 'Unable to write log record to file (error code 0x%X)', arg1 := F_UDINT(fbFilePuts.nErrId), sOut => sFaultDescription);
				eState := E_LogToDiskState.Error;
			ELSE // Done, write the log message
				eState := E_LogToDiskState.WriteLogItemMessage;
			END_IF
		END_IF
	
	E_LogToDiskState.WriteLogItemMessage:
		IF fbStateMachine.bStateChanged THEN
			fbFilePuts.sLine := CONCAT(stLogItemToDisk.sMsg, '$L'); // Add line feed character
		END_IF
		fbFilePuts(bExecute := TRUE, hFile := fbFileOpen.hFile);
		IF (NOT fbFilePuts.bBusy) THEN
			fbFilePuts(bExecute := FALSE);
			IF fbFilePuts.bError THEN
				fbFormatString(sFormat := 'Unable to write log record to file (error code 0x%X)', arg1 := F_UDINT(fbFilePuts.nErrId), sOut => sFaultDescription);
				eState := E_LogToDiskState.Error;
			ELSE // Done, get the next log item in the buffer
				IF (stLogItemFromBuffer.sMsg <> '') THEN 
					// Last log item retrieved from the buffer wasn't written yet (e.g., after new file creation), so no need to pop items from the buffer yet
					eState := E_LogToDiskState.CloseFile;
				ELSE // Check if there are more items in the buffer
					stLogItemFromBuffer := Pop();
					IF (stLogItemFromBuffer.sMsg = '') THEN // Buffer empty, close the file
						eState := E_LogToDiskState.CloseFile;
					ELSE // More items to be written, but first check file size before adding more items
						eState := E_LogToDiskState.CheckFileSize;
					END_IF
				END_IF
			END_IF
		END_IF
	
	E_LogToDiskState.CloseFile:
		fbFileClose(bExecute := TRUE, hFile := fbFileOpen.hFile);
		IF (NOT fbFileClose.bBusy) THEN
			fbFileClose(bExecute := FALSE);
			IF fbFileClose.bError THEN
				fbFormatString(sFormat := 'Unable to close file (error code 0x%X)', arg1 := F_UDINT(fbFileClose.nErrId), sOut => sFaultDescription);
				eState := E_LogToDiskState.Error;
			ELSE
				eState := E_LogToDiskState.FindObsoleteFiles;
			END_IF
		END_IF
	
	E_LogToDiskState.FindObsoleteFiles:
		// Delete oldest log files in log folder until we're at MAX_NUMBER_OF_LOG_FILES
		IF fbStateMachine.bStateChanged THEN
			nFileCount := 0;	
			tOldestLogFile.sFileName := ''; 
			// Create a path search string, e.g. '/tmp/Log_*.txt'
			fbFormatString(
				sFormat := '%s%s*.%s',
				arg1 := F_STRING(sLogFolder),
				arg2 := F_STRING(sLogFilePrefix),
				arg3 := F_STRING(sLogFileExtension),
				sOut => fbEnumFiles.sPathName
			);
			fbEnumFiles.eCmd := E_EnumCmdType.eEnumCmd_First;
		END_IF
		fbEnumFiles(bExecute := TRUE);
		IF (NOT fbEnumFiles.bBusy) THEN
			fbEnumFiles(bExecute := FALSE, eCmd := E_EnumCmdType.eEnumCmd_Next);
			IF fbEnumFiles.bError THEN
				fbFormatString(
					sFormat := 'Unable to get files in folder "%s" (error code 0x%X)',
					arg1 := F_STRING(fbEnumFiles.sPathName),
					arg2 := F_UDINT(fbEnumFiles.nErrId),
					sOut => sFaultDescription
				);
				eState := E_LogToDiskState.Error;
			ELSIF fbEnumFiles.bEOE THEN
				// Found all files, carry on
				eState := E_LogToDiskState.WaitForCommand;
				bLoggerInitialized := TRUE;
			ELSE
				// Found a file, check if it's older than the previous find
				nFileCount := nFileCount + 1;
				IF (tOldestLogFile.sFileName = '') 
					OR (PLWORD_TO_LWORD(ADR(fbEnumFiles.stFindFile.creationTime)) < PLWORD_TO_LWORD(ADR(tOldestLogFile.creationTime))) 
				THEN
					tOldestLogFile := fbEnumFiles.stFindFile;
				END_IF
				IF (nFileCount > nMaxNumberOfLogFiles) THEN
					// Max number of log files reached, delete the file				
					eState := E_LogToDiskState.DeleteFile;
				END_IF
			END_IF
		END_IF

	E_LogToDiskState.DeleteFile:
		IF fbStateMachine.bStateChanged THEN
			fbFormatString(
				sFormat := '%s%s',
				arg1 := F_STRING(sLogFolder),
				arg2 := F_STRING(tOldestLogFile.sFileName),
				sOut => fbFileDelete.sPathName
			);
		END_IF
		fbFileDelete(bExecute := TRUE);
		IF (NOT fbFileDelete.bBusy) THEN
			fbFileDelete(bExecute := FALSE);
			IF fbFileDelete.bError THEN
				fbFormatString(
					sFormat := 'Unable to delete file "%s" (error code 0x%X)',
					arg1 := F_STRING(tOldestLogFile.sFileName),
					arg2 := F_UDINT(fbFileClose.nErrId), 
					sOut => sFaultDescription
				);
				eState := E_LogToDiskState.Error;
			ELSE // Done deleting, continue searching for obsolete files
				eState := E_LogToDiskState.FindObsoleteFiles;
			END_IF
		END_IF

	E_LogToDiskState.Error:
		IF (sFaultDescription = '') THEN
			sFaultDescription := 'Unknown error';
		END_IF

END_CASE

bFault S= (eState = E_LogToDiskState.Error);

METHOD INTERNAL FINAL AddToLog
VAR_INPUT
	stLogItem : UDT_LogItem;
END_VAR
VAR
	bOk : BOOL;
	nMaxItems : UDINT;
END_VAR
// Ignore incoming items when the logger has an error
IF bFault THEN
	RETURN;
END_IF


fbBuffer.A_AddTail(
	pWrite := ADR(stLogItem),
	cbWrite := SIZEOF(stLogItem),
	bOk => bOk,
);

IF NOT bOk THEN // Buffer overflow
	// Make sure no more items will be added to the log
	bFault := TRUE;
	// Pop last item to make room for the famous last words
	Pop(); 
	// And add those words to the log
	nMaxItems := MAX_ITEMS_IN_BUFFER;
	fbFormatString(
		sFormat := 'Log buffer size limit (%u) reached! Dumping buffer and disabling the log handler.',
		arg1 := F_UDINT(nMaxItems),
		sOut => sFaultDescription
	);
	stLogItem.sMsg := sFaultDescription;
	stLogItem.eLevel := E_LogLevel.FATAL;
	fbBuffer.A_AddTail(
		pWrite := ADR(stLogItem),
		cbWrite := SIZEOF(stLogItem),
		bOk => bOk,
	);
END_IF
END_METHOD

METHOD PROTECTED CreatePath : STRING // Create a filename with a date/time stamp, e.g. "/tmp/Log_20230203-093610.txt'
VAR
	fMonth : REAL;
	fDay : REAL;
	fHour : REAL;
	fMinute : REAL;
	fSecond : REAL;
END_VAR
// Suppress error "VAR_IN_OUT parameter 'in' needs variable with write access as input."	
fMonth := WORD_TO_REAL(Sys_Variables.SystemTime_TS.wMonth); 
fDay := WORD_TO_REAL(Sys_Variables.SystemTime_TS.wDay); 
fHour := WORD_TO_REAL(Sys_Variables.SystemTime_TS.wHour); 
fMinute := WORD_TO_REAL(Sys_Variables.SystemTime_TS.wMinute); 
fSecond := WORD_TO_REAL(Sys_Variables.SystemTime_TS.wSecond); 

fbFormatString(
	sFormat := '%s%s%u%02.0f%02.0f-%02.0f%02.0f%02.0f.%s',
	arg1 := F_STRING(sLogFolder),
	arg2 := F_STRING(sLogFilePrefix),
	arg3 := F_WORD(Sys_Variables.SystemTime_TS.wYear),
	arg4 := F_REAL(fMonth),
	arg5 := F_REAL(fDay),
	arg6 := F_REAL(fHour),
	arg7 := F_REAL(fMinute),
	arg8 := F_REAL(fSecond),
	arg9 := F_STRING(sLogFileExtension),
	sOut => CreatePath
);
END_METHOD

METHOD FB_init : BOOL
VAR_INPUT
	bInitRetains : BOOL; // if TRUE, the retain variables are initialized (warm start / cold start)
	bInCopyCode : BOOL;  // if TRUE, the instance afterwards gets moved into the copy code (online change)

	sLogFolder 			: T_MaxString; // Example for TwinCAT/BSD: '/tmp/'. The folder where log files will be stored. Add trailing '/' or '\'. 
	sLogFilePrefix 		: T_MaxString; // Example: 'Log_'
	sLogFileExtension 	: T_MaxString; // Example: 'txt'
	nMaxLogFileSize 	: ULINT; // [bytes] When this size is reached, a new log file is created 
	nMaxNumberOfLogFiles: UINT;
END_VAR
THIS^.sLogFolder := sLogFolder;
IF (sLogFolder = '') THEN
	bFault := TRUE;
	sFaultDescription := 'Parameter "sLogFolder" empty';
END_IF
THIS^.sLogFilePrefix := sLogFilePrefix;
THIS^.sLogFileExtension := sLogFileExtension;
THIS^.nMaxLogFileSize := nMaxLogFileSize;
THIS^.nMaxNumberOfLogFiles := nMaxNumberOfLogFiles;
END_METHOD

METHOD PROTECTED Pop : UDT_LogItem; // Pops the buffer head (returns the oldest log item in the buffer)
fbBuffer.A_RemoveHead(
	pRead:= ADR(Pop),
	cbRead:= SIZEOF(Pop),
);
END_METHOD

END_FUNCTION_BLOCK

// ---- Logger/Functions/LogHandlers/FB_LogHandlerBase.TcPOU
{attribute 'reflection'}
FUNCTION_BLOCK PUBLIC ABSTRACT FB_LogHandlerBase // Base class for all log handlers
VAR_OUTPUT
	{attribute 'instance-path'} 
    {attribute 'noinit'}
	sInstancePath : STRING; // Instance path of the function block
END_VAR

METHOD INTERNAL ABSTRACT AddToLog
VAR_INPUT
	stLogItem : UDT_LogItem;
END_VAR
END_METHOD

END_FUNCTION_BLOCK

// ---- Logger/Functions/LogHandlers/FB_LogHandler_ADSLOG.TcPOU
FUNCTION_BLOCK FB_LogHandler_ADSLOG EXTENDS FB_LogHandlerBase // Writes log item to the ADS log
VAR
END_VAR

METHOD INTERNAL FINAL AddToLog
VAR_INPUT
	stLogItem : UDT_LogItem;
END_VAR
VAR
	msgCtrlMask : DWORD; // ADS log message control mask, more info: https://infosys.beckhoff.com/content/1033/tcplclib_tc2_system/31030539.html	
END_VAR
msgCtrlMask := ADSLOG_MSGTYPE_LOG OR ADSLOG_MSGTYPE_STRING;
CASE stLogItem.eLevel OF
	E_LogLevel.TRACE: 	msgCtrlMask := msgCtrlMask OR ADSLOG_MSGTYPE_HINT;
	E_LogLevel.DEBUG: 	msgCtrlMask := msgCtrlMask OR ADSLOG_MSGTYPE_HINT;
	E_LogLevel.INFO: 	msgCtrlMask := msgCtrlMask OR ADSLOG_MSGTYPE_HINT;
	E_LogLevel.WARN: 	msgCtrlMask := msgCtrlMask OR ADSLOG_MSGTYPE_WARN;
	E_LogLevel.ERROR:	msgCtrlMask := msgCtrlMask OR ADSLOG_MSGTYPE_ERROR;
	E_LogLevel.FATAL: 	msgCtrlMask := msgCtrlMask OR ADSLOG_MSGTYPE_ERROR;
END_CASE

ADSLOGSTR(
	msgCtrlMask := msgCtrlMask,
	msgFmtStr := '%s',
	strArg := stLogItem.sMsg
);
END_METHOD

END_FUNCTION_BLOCK

// ---- Logger/Functions/FB_Logger.TcPOU
FUNCTION_BLOCK PUBLIC FB_Logger
VAR_STAT
	aLogHandlers : ARRAY[1..10] OF UDT_LogHandlerConfig; // The log handlers that process the incoming log messages
	bUnexpectedCall : BOOL; // FB_Logger should never be called. Use this bit to avoid flooding the log.
END_VAR

IF NOT bUnexpectedCall THEN
	THIS^.FATAL('Unexpected call to FB_Logger(). Do not call FB_Logger!');
	bUnexpectedCall := TRUE;
END_IF

METHOD PUBLIC DEBUG // Add a message to the log with log level DEBUG 
(*
The DEBUG level is used for logging messages that help developers find out what went wrong
during a debugging session. While the specifics of what messages to log at the DEBUG level
is dependent on your application, you generally want to include detailed information that
can help developers troubleshoot an issue quickly. 
This can include variable state in the surrounding scope, or relevant error codes.
Unlike TRACE, DEBUG level logging can be turned on in production without making the application unusable,
but it should not be left on indefinitely to ensure the log is not flooded.
*)
VAR_INPUT
	sMsg : T_MaxString; // The message to be logged
END_VAR
THIS^.SendToLogHandlers(sMsg, E_LogLevel.DEBUG);
END_METHOD

METHOD PUBLIC ERROR // Add a message to the log with log level ERROR
(*
The ERROR log level is used to represent error conditions in a system that
prevent a specific operation from running, but the system itself can continue
working even if it is at a reduced level of functionality or performance.
Generally, ERROR logs should be investigated as soon as possible but they don't
carry the same urgency as FATAL messages since the system can continue working.
*)
VAR_INPUT
	sMsg : T_MaxString; // The message to be logged
END_VAR
THIS^.SendToLogHandlers(sMsg, E_LogLevel.ERROR);
END_METHOD

METHOD PUBLIC FATAL // Add a message to the log with log level FATAL
(*
The FATAL log level annotates messages with the greatest severity.
It usually means that something critical is broken, and the system cannot continue to do any more
useful work without the intervention of an engineer. T
ypically, such entries are logged before the system is shut down ("famous last words").
*)
VAR_INPUT
	sMsg : T_MaxString; // The message to be logged
END_VAR
THIS^.SendToLogHandlers(sMsg, E_LogLevel.FATAL);
END_METHOD

METHOD PUBLIC INFO // Add a message to the log with log level INFO
(*
INFO-level messages indicate events in the system that are significant to the
general purpose of the system. Such events are logged to show that the system is
operating normally. For example, a recipe was started or stopped. 
Production systems typically default to logging at this level so that a 
summary of the application's normal behavior is visible to anyone reading the logs.
*)
VAR_INPUT
	sMsg : T_MaxString; // The message to be logged
END_VAR
THIS^.SendToLogHandlers(sMsg, E_LogLevel.INFO);
END_METHOD

METHOD PUBLIC RegisterLogHandler : BOOL
VAR_IN_OUT
	fbLogHandler : FB_LogHandlerBase;
END_VAR
VAR_INPUT
	eMinimumLogLevel : E_LogLevel;
END_VAR
VAR
	i : USINT; // Iterator
END_VAR
RegisterLogHandler := TRUE;
FOR i := 1 TO 10 DO
	IF aLogHandlers[i].pLogHandler = ADR(fbLogHandler) THEN // Already added
		RETURN;
	ELSIF aLogHandlers[i].pLogHandler = 0 THEN // Found empty spot in the array, add the log handler
		aLogHandlers[i].pLogHandler := ADR(fbLogHandler);
		aLogHandlers[i].eMinimumLogLevel := eMinimumLogLevel;
		RegisterLogHandler := TRUE;
		DEBUG(CONCAT('Added log handler: ', fbLogHandler.sInstancePath));
		RETURN;
	END_IF
END_FOR
RegisterLogHandler := FALSE; // Failed to add loghandler
END_METHOD

METHOD PUBLIC Run // Enables the logger and log handlers, should be called once every PLC cycle in your program/project (not multiple calls per cycle!)
VAR
	i : USINT; // Iterator
END_VAR
// Call every log handler. Only relevant for log handlers that take multiple PLC cycles
// to handle incoming log items (e.g., writing log items to disk).
FOR i := 1 TO 10 DO
	IF aLogHandlers[i].pLogHandler <> 0 THEN
		aLogHandlers[i].pLogHandler^();
	END_IF
END_FOR
END_METHOD

METHOD PRIVATE SendToLogHandlers
VAR_INPUT
	sMsg : T_MaxString; // The message to be logged
	eLevel : E_LogLevel; // Log level (debug, info, warn, etc.)
END_VAR
VAR
	stLogItem : UDT_LogItem;
	i : USINT; // Iterator
END_VAR
// Ignore empty messages
IF (sMsg = '') THEN
	RETURN;
END_IF

// Create a log item
stLogItem.sMsg := sMsg;
stLogItem.eLevel := eLevel;
stLogItem.stTimestamp := Sys_Variables.SystemTime_TS;

// Add item to all registered loghandlers (if level is high enough)
FOR i := 1 TO 10 DO
	IF (aLogHandlers[i].pLogHandler <> 0) AND (eLevel >= aLogHandlers[i].eMinimumLogLevel) THEN
		aLogHandlers[i].pLogHandler^.AddToLog(stLogItem);
	END_IF
END_FOR
END_METHOD

METHOD PUBLIC TRACE // Add a message to the log with log level TRACE
(*
The TRACE level can be used for tracing the path of code execution in a program.
Generally, TRACE is used for showing the flow of the program, and to provide a detailed breakdown of the sequence
of events that led to a crash, a silent failure, an error, or some other event logged at a different level.
The TRACE level is only used temporarily (when the code is a "work in progress").
*)
VAR_INPUT
	sMsg : T_MaxString; // The message to be logged
END_VAR
THIS^.SendToLogHandlers(sMsg, E_LogLevel.TRACE);
END_METHOD

METHOD PUBLIC WARN // Add a message to the log with log level WARN
(*
Messages logged at the WARN level typically indicate that something unexpected happened,
but the system can recover and continue to function normally.
It is mainly used to draw attention to situations that should be addressed soon before
they pose a problem for the system.
*)
VAR_INPUT
	sMsg : T_MaxString; // The message to be logged
END_VAR
THIS^.SendToLogHandlers(sMsg, E_LogLevel.WARN);
END_METHOD

END_FUNCTION_BLOCK

// ---- System/Functions/DataManagement/FB_PersistentDataManager.TcPOU
FUNCTION_BLOCK FB_PersistentDataManager
VAR_INPUT
END_VAR
VAR_OUTPUT
END_VAR
VAR
	FbWritePersistentData : FB_WritePersistentData ;
	cmdWrite : BOOL := FALSE ;
	TOfWriteInterval	: TOf ;
	CmdWriteFromTime	: BOOL ; 
	TestjeWritten		: BOOL ;
END_VAR

// ===== persistent write interval =====
 TOfWriteInterval(	IN := cmdWrite OR NOT TOfWriteInterval.Q,
	 				PT	:= T#5M  );

IF NOT TOfWriteInterval.Q THEN 
	cmdWrite := TRUE ;
END_IF

// ===== write persistent data =====
	FbWritePersistentData ( PORT 	:= 851,
							START 	:= CmdWrite,
							TMOUT 	:= T#1S,	
							mode 	:= E_PersistentMode.SPDM_VAR_BOOST );	

IF cmdWrite AND FbWritePersistentData.BUSY THEN 
	cmdWrite := FALSE ;
END_IF

METHOD PUBLIC Write : BOOL
VAR_INPUT
END_VAR
IF NOT FbWritePersistentData.BUSY THEN 
	cmdWrite := TRUE ;
ELSE 
	Write := TRUE ;
END_IF
END_METHOD

END_FUNCTION_BLOCK

// ---- FaultsAndMessages/Functions/FB_FaultHandler.TcPOU
FUNCTION_BLOCK FB_FaultHandler
(* 
The faulthandler is responsible for 
	- providing the means for objects to register their faults
	- reporting the active fault types (i.e., message, fatal fault, etc.) --> arActiveFaultTypes
	- providing the means to reset a fault type
	- keeping a log of all faults

It is not responsible for
	- resetting the actual fault (this is up to the object that registered the fault)
	- handling any HMI related functionality

Active faults do not disappear from the log, the need to be manually cleared by issuing a CmdReset and CmdClearInactive.
*)
VAR_INPUT
	nMaxInactiveCycles : UINT := 50; // Once faults haven't been activated for a number of PLC cycles, deactivate them. 0 = do not automatically deactivate faults 
END_VAR
VAR_OUTPUT
	arFaultLog 			: ARRAY [1..PAR_Utilities.MAX_FAULTS_IN_LOG] OF UDT_FaultLogItem;
	nFaultsInLog 		: UINT;
	nActiveFaults 		: UINT;
	arActiveFaultTypes 	: ARRAY[0..(E_FaultTypes._ENUM_SIZE - 1)] OF BOOL; // Status of each fault type
END_VAR
VAR
	fbLogger : FB_Logger;

	bCmdReset : BOOL;
	eResetState : E_ResetState;
	arActiveFaultTypes_Internal : ARRAY[0..(E_FaultTypes._ENUM_SIZE - 1)] OF BOOL; // The actual status of each fault type, which is reported unless the reset cycle is active
	
	nLogIndex : UINT; // Array index of the last added item in the log (zero until the first item arrives)
	nIterIndex : UINT; // Index of the fault log iterator (used for properties First and Next)

	fbFormatString : FB_FormatString; // https://infosys.beckhoff.com/content/1033/tcplclib_tc2_utilities/34990219.html
END_VAR

UpdateInactiveCycles();

ExecReset();

UpdateActiveFaultStatus();

METHOD PROTECTED AddFaultToLog
VAR_INPUT
	stFaultLogItem : UDT_FaultLogItem;
	bActivated : BOOL; // TRUE means the fault has just been activated, FALSE means it stopped being active
END_VAR
VAR
	sStatus : T_MaxString;
	sFaultType : T_MaxString;
	sId : T_MaxString;
	sDescription : T_MaxString;
	sMsg : T_MaxString;
END_VAR
IF bActivated THEN
	sStatus := 'START';
ELSE
	sStatus := 'END';
END_IF
sFaultType := TO_STRING(stFaultLogItem.stFault.FaultType);
sId := stFaultLogItem.Id;
sDescription := stFaultLogItem.stFault.Description;

fbFormatString(
	sFormat := '[%s %s] %s - %s',
	arg1 := F_STRING(sFaultType),
	arg2 := F_STRING(sStatus),
	arg3 := F_STRING(sId),
	arg4 := F_STRING(sDescription),
	sOut => sMsg
);

CASE stFaultLogItem.stFault.FaultType OF
	E_FaultTypes.OM: fbLogger.INFO(sMsg); 
	E_FaultTypes.OW: fbLogger.WARN(sMsg); 
	E_FaultTypes.MC: fbLogger.WARN(sMsg); 
	E_FaultTypes.CF: fbLogger.WARN(sMsg); 
	E_FaultTypes.FF: fbLogger.ERROR(sMsg); 
END_CASE
END_METHOD

METHOD PUBLIC CmdAddFault : BOOL
(*
CmdAddFault should be called every cycle.
If the fault is active, it's corresponding fault type is enabled.
Updates the fault log.
*)
VAR_IN_OUT
	stFault : UDT_Fault; // active fault structure input
END_VAR
VAR_INPUT
	stIdentity : UDT_Identity;
END_VAR
// Update the log
UpdateLog(stFault, stIdentity);

// Clear active status (to be updated by caller)
stFault.Active := FALSE;
END_METHOD

METHOD PUBLIC CmdClearInactive : BOOL // Remove inactive faults from the log
VAR
	stEmptyItem : UDT_FaultLogItem;
	i : UINT; // Iterator
END_VAR
nFaultsInLog := PAR_Utilities.MAX_FAULTS_IN_LOG;
IF (eResetState = E_ResetState.Idle) THEN
	FOR i := 1 TO PAR_Utilities.MAX_FAULTS_IN_LOG DO
		IF (NOT arFaultLog[i].stFault.Active) THEN
			nFaultsInLog :=nFaultsInLog - 1;
			arFaultLog[i] := stEmptyItem;
			arFaultLog[i].bEmpty := TRUE;
		END_IF
	END_FOR
	CmdClearInactive := TRUE;
ELSE
	CmdClearInactive := FALSE;
END_IF
END_METHOD

METHOD PUBLIC CmdReset : BOOL // Reset faults; caller is responsible for stopping the call once TRUE is returned
VAR_INPUT
END_VAR
// Trigger the reset cycle
IF (eResetState = E_ResetState.Idle) THEN
	bCmdReset := TRUE;
END_IF

CmdReset := (eResetState = E_ResetState.Done); // Let the caller know when the reset cycle is finished
END_METHOD

METHOD PRIVATE ExecReset : BOOL
VAR
	i : UINT; // Iterator
END_VAR
CASE eResetState OF
	E_ResetState.Idle: // Wait for reset command
		IF bCmdReset THEN
			// Start the reset cycle
			bCmdReset := FALSE;
			eResetState := E_ResetState.ResetFaultTypes;
		ELSE
			ReportActiveFaultStatus();
		END_IF
	E_ResetState.ResetFaultTypes: 
		// During a reset, the active fault types are not updated 
		// This avoids that faults are not reported for 1 PLC cycle, even though they are still active
		// We do however clear the internal fault types, which are updated automatically during the WaitForFaults state.
		FOR i:= 0 TO (E_FaultTypes._ENUM_SIZE - 1) DO		
			arActiveFaultTypes_Internal[i] := FALSE;
		END_FOR
		eResetState := E_ResetState.WaitForFaults;

	E_ResetState.WaitForFaults: // Allow the PLC one cycle to re-add faults
		eResetState := E_ResetState.Done;

	E_ResetState.Done: // Done, report & allow caller one cycle to reset itself
		ReportActiveFaultStatus();
		eResetState := E_ResetState.Idle;
END_CASE
END_METHOD

METHOD PRIVATE FindNonEmptyFault : UINT // Update nIterIndex to first non-empy fault (if available)
VAR_INPUT
	nStartIndex : UINT;
END_VAR
VAR
	i : UINT; // Iterator
END_VAR
// Sanitize input
IF nStartIndex = 0 THEN
	nStartIndex := PAR_Utilities.MAX_FAULTS_IN_LOG;
ELSE
	nStartIndex := MIN(nStartIndex, PAR_Utilities.MAX_FAULTS_IN_LOG);
END_IF

// Iterate array backwards until a non empty item is found.
FOR i := 1 TO PAR_Utilities.MAX_FAULTS_IN_LOG DO
	IF arFaultLog[nStartIndex].bEmpty THEN
		nStartIndex := nStartIndex - 1;
		IF nStartIndex = 0 THEN
			nStartIndex := PAR_Utilities.MAX_FAULTS_IN_LOG;
		END_IF
	ELSE
		EXIT;
	END_IF
END_FOR

FindNonEmptyFault := nStartIndex;
END_METHOD

PROPERTY PUBLIC Head : UDT_FaultLogItem // Returns the head of the log (the latest item added)
GET
nIterIndex := FindNonEmptyFault(nLogIndex);
Head := arFaultLog[nIterIndex];
END_GET
SET
END_SET
END_PROPERTY

PROPERTY PUBLIC Next : UDT_FaultLogItem // Get the next item in the log (travelling backwards through the array)
GET
nIterIndex := FindNonEmptyFault(nIterIndex - 1);
Next := arFaultLog[nIterIndex];
END_GET
SET
END_SET
END_PROPERTY

METHOD PRIVATE ReportActiveFaultStatus : BOOL // Update active fault types based on active faults in the log
VAR
	i : UINT; // Iterator
END_VAR
// Report the status of each fault type to outside world	
FOR i:= 0 TO (E_FaultTypes._ENUM_SIZE - 1) DO		
	arActiveFaultTypes[i] := arActiveFaultTypes_Internal[i];
END_FOR
END_METHOD

METHOD PRIVATE UpdateActiveFaultStatus : BOOL // Update active fault types based on active faults in the log
VAR
	i : UINT; // Iterator
END_VAR
// Get active faults from log
nActiveFaults := 0;
FOR i := 1 TO PAR_Utilities.MAX_FAULTS_IN_LOG DO
	IF (arFaultLog[i].stFault.Active) THEN 
		// Update the number of active faults
		nActiveFaults := nActiveFaults + 1;
		// Update active fault type feedback
		arActiveFaultTypes_Internal[arFaultLog[i].stFault.FaultType] := TRUE; 
	END_IF
END_FOR
END_METHOD

METHOD PRIVATE UpdateInactiveCycles : BOOL // Update the number of inactive cycles, and deactive fault once it reaches the max number of inactive cycles
VAR
	i : UINT; // Iterator
END_VAR
IF (nMaxInactiveCycles > 0) THEN
	FOR i := 1 TO PAR_Utilities.MAX_FAULTS_IN_LOG DO
		IF arFaultLog[i].stFault.Active THEN
			arFaultLog[i].nInactiveCycles := MIN(16#FFFF, arFaultLog[i].nInactiveCycles + 1);
			IF (arFaultLog[i].nInactiveCycles > nMaxInactiveCycles) THEN
				arFaultLog[i].stFault.Active := FALSE;
				arFaultLog[i].EndTime := Sys_Variables.SystemTime;	
			END_IF
		END_IF
	END_FOR
END_IF
END_METHOD

METHOD PRIVATE UpdateLog : BOOL
(*
Update the fault log array. 
If a fault becomes active, it is added to the array and the start time is updated.
If a fault stops being active, the end time is updated.
Inactive faults are cleared by CmdReset.
*)
VAR_IN_OUT
	stFault : UDT_Fault;
END_VAR
VAR_INPUT
	stIdentity : UDT_Identity;
END_VAR
VAR
	sId : STRING;
	nFaultIndexInLog : UINT;
	i : UINT; // Iterator
END_VAR
// Check if the fault already exists in the log. 
// For this, we need to compare the description and the fault ID.

// First, build the fault ID
sId := TO_STRING(stFault.FaultType);
sId := CONCAT(sId,'.');
IF stIdentity.nParentId > 0 THEN
	sId := CONCAT(sId,UDINT_TO_STRING(stIdentity.nParentId));
	sId := CONCAT(sId,'.');
END_IF
sId := CONCAT(sId,UINT_TO_STRING(stIdentity.nId));
sId := CONCAT(sId,'.');
sId := CONCAT(sId,UDINT_TO_STRING(stIdentity.eComponentType));
sId := CONCAT(sId,'.');
sId := CONCAT(sId,stIdentity.sName);

// Now check if the fault already exists in the log
FOR i := 1 TO PAR_Utilities.MAX_FAULTS_IN_LOG DO
	IF (NOT arFaultLog[i].bEmpty) 
		AND (arFaultLog[i].Id = sId) 
		AND (arFaultLog[i].stFault.Description = stFault.Description)
		AND (ANY_TO_DWORD(arFaultLog[i].EndTime) = 0)
	THEN // Found fault in the log
		nFaultIndexInLog := i;
		EXIT; // No need to iterate any further
	END_IF
END_FOR

IF nFaultIndexInLog > 0 THEN // Already exists in the log
	IF (stFault.Active) THEN // Still active, reset inactive cycle counter
		arFaultLog[nFaultIndexInLog].nInactiveCycles := 0;
	ELSIF (ANY_TO_DWORD(arFaultLog[nFaultIndexInLog].EndTime) = 0) THEN // No longer active, update end time and active state
		arFaultLog[nFaultIndexInLog].stFault.Active := FALSE;
		arFaultLog[nFaultIndexInLog].EndTime := Sys_Variables.SystemTime;
		AddFaultToLog(arFaultLog[nLogIndex], FALSE);
	END_IF
ELSIF stFault.Active THEN // New active fault, add it to the log
	// Update the log index (if full, move to beginning of the log)
	nLogIndex := (nLogIndex MOD PAR_Utilities.MAX_FAULTS_IN_LOG) + 1;
	nFaultsInLog := MIN(nFaultsInLog + 1, PAR_Utilities.MAX_FAULTS_IN_LOG);
	// Copy to log and update start time
	arFaultLog[nLogIndex].bEmpty := FALSE;
	arFaultLog[nLogIndex].stFault := stFault;
	arFaultLog[nLogIndex].Id := sId;
	arFaultLog[nLogIndex].StartTime := Sys_Variables.SystemTime;
	arFaultLog[nLogIndex].EndTime := ANY_TO_DT(0);
	arFaultLog[nLogIndex].nInactiveCycles := 0;
	AddFaultToLog(arFaultLog[nLogIndex], TRUE);
END_IF
END_METHOD

END_FUNCTION_BLOCK

// ---- System/Functions/Fb_SystemVariables.TcPOU
FUNCTION_BLOCK Fb_SystemVariables
VAR
	// **** Function blocks *****
		Fb_SystemTime: FB_LocalSystemTime ;
		Fb_TimerHbOn : Ton ; // Timer Heartbeat on
		Fb_TimerFast : Ton ; // Timer for fast blink bit
		Fb_TimerSlow : Ton ; // Timer for slow blink bit
		Fb_RisingPulse : R_Trig ; // Rinsing edge trigger function	
	// ***** internal Variables *****
		HeartbeatOn	: BOOL ; // heartbeat is on
		FlashFastOn	: BOOL ; // Fast Flash bit on
		FlashSlowOn	: BOOL ; // Flash slow bit on
	
		Fb_Timer100mSec : TON := (PT := T#100MS); // Timer for 100 ms pulse
		
		fbFormatString : FB_FormatString;
END_VAR

// ===== Get system time =====
	// ***** get windows system time *****
		Fb_SystemTime(	sNetID := '', 
						bEnable := TRUE, 
						dwCycle := 1,
						dwOpt := 0, 
						tTimeout := DEFAULT_ADS_TIMEOUT, 	
						systemTime => Sys_Variables.SystemTime_TS,
						tzID	=> Sys_Variables.TimeZoneId
						);
	// ****** convert to time of day format *****
		Sys_Variables.SystemTime := SYSTEMTIME_TO_DT(TIMESTR := Sys_Variables.SystemTime_TS) ;
		
// ===== Heartbeat generator =====
	Fb_TimerHbOn(In := NOT HeartbeatOn , PT:= T#1S, Q => HeartbeatOn);
	IF Fb_TimerHbOn.ET >= T#500MS THEN
		Sys_Variables.HeartBeat := TRUE ;
	ELSE
		Sys_Variables.HeartBeat := FALSE ;
	END_IF

// ===== one second pulse generator =====
	Fb_RisingPulse(Clk := HeartbeatOn, Q => Sys_Variables.Pulse1Sec);
	
// ===== 100ms pulse generation ======
	Fb_Timer100mSec( IN := NOT Sys_Variables.Pulse100ms, Q => Sys_Variables.Pulse100ms);

// ===== Flash fast bit =====
	Fb_TimerFast(In := NOT FlashFastOn, Pt := T#1S, Q => FlashFastOn);
	IF Fb_TimerFast.ET >= T#600MS THEN
		Sys_Variables.BlinkFast := TRUE;  
	ELSE
		Sys_Variables.BlinkFast := FALSE;  		
	END_IF
// ===== Flash Slow bit =====
	Fb_TimerSlow(In := NOT FlashSLowOn, Pt := T#2S, Q => FlashSlowOn);
	IF Fb_TimerSlow.ET >= T#1200MS THEN
		Sys_Variables.BlinkSlow := TRUE;  
	ELSE
		Sys_Variables.BlinkSlow := FALSE;  		
	END_IF

// ===== Always true and always false bits =====
	Sys_Variables.AlwaysOff := FALSE 	;
	Sys_Variables.AlwaysOn	:= TRUE		;
	
// ===== Manage persistent data ======
	DataManager.FbPersistentManager();

END_FUNCTION_BLOCK

// ---- BaseFunctions/FB_FunctionBase.TcPOU
{attribute 'reflection'}
FUNCTION_BLOCK PUBLIC ABSTRACT FB_FunctionBase EXTENDS FB_Base
VAR_OUTPUT
	sActiveState	: STRING 		:= 'Idle'	; // active state of device 
	bManual			: BOOL 			:= FALSE 	; // device is in manual mode
	bIsSafe			: BOOL 			:= FALSE	; // Device is locked and safe
	bHeld			: BOOL 			:= FALSE 	; // Function is held
	bBlockedCommand	: BOOL 			:= FALSE 	; // a device command is blocked because of collision detect 
END_VAR
VAR
	bCmdManual 		: BOOL			:= FALSE	; // manual commands enabled control functions (thus disable automatic)
END_VAR

SUPER^();

// Communicate active state
IF bErrorActive THEN 
	sActiveState := TO_STRING(stFault.Description);
ELSIF NOT bInitOk THEN 
	sActiveState := 'Not initialized';
ELSIF bManual THEN 
	sActiveState := 'Manual operation';
ELSE
	sActiveState := 'Operational';
END_IF 

// Set manual command mode
bManual := bCmdManual;

// Execute device functions
IF bInitOk THEN  
	ExecMachineSafety();
	ExecDevFunctions();
END_IF

// Set fault if commands are blocked
IF bBlockedCommand AND bHeld THEN 
	stFault.Active 			:= TRUE ;
	stFault.Description		:= 'Function is blocked';
	stFault.FaultType		:= E_FaultTypes.MC;
END_IF

METHOD PUBLIC CmdHold : BOOL
VAR_INPUT
END_VAR
bHeld 	:= TRUE ;
CmdHold := bHeld ;
END_METHOD

METHOD PUBLIC CmdManual : BOOL
VAR_INPUT
END_VAR
// Enable manual mode
bCmdManual := TRUE;
END_METHOD

METHOD PUBLIC CmdSafeStop : BOOL
VAR_INPUT
END_VAR
// check if device is safe
bIsSafe 	:= NOT bEnable ;
CmdSafeStop := bIsSafe ;
END_METHOD

METHOD PROTECTED ExecDevFunctions : BOOL
VAR_INPUT
END_VAR
END_METHOD

METHOD PROTECTED ExecMachineSafety : BOOL
VAR_INPUT
END_VAR
END_METHOD

END_FUNCTION_BLOCK

// ---- Compare/Functions/Between.TcPOU
FUNCTION Between : BOOL // Returns true if value is >= the lower and <= the upper threshold
VAR_INPUT
	Lower	: LREAL	; // lower threshold value [LREAL]
	Value	: LREAL	; // test value [LREAL]
	Upper	: LREAL	; // Upper threshold value [LREAL]
END_VAR
VAR
END_VAR

// Check if value is between lower and upper threshold
Between := (Value >= Lower) AND (Value <= Upper);

END_FUNCTION

// ---- Conversion/DegS_To_Rpm_And_MMin.TcPOU
FUNCTION DegS_To_Rpm_And_MMin : BOOL
VAR_INPUT
	DegPerSecond : LREAL ; // Input degrees per second
	StitchLength : LREAL ; // Input stitch length
END_VAR
VAR_OUTPUT
	RevPerMinute	: LREAL ; // Output revolutions per minute
	MetersPerMinute	: LREAL ; // Output meters per minute
END_VAR
VAR
END_VAR

// ===== convert degrees per second to Rpm =====
	RevPerMinute := (DegPerSecond/360)*60 ;
// ===== Convert RPM to MMin =====
	MetersPerMinute := RevPerMinute * StitchLength / 1000 ;

END_FUNCTION

// ---- Conversion/Grey_To_Bin.TcPOU
FUNCTION Grey_To_Bin : INT // convert 4 bit grey code into 8 bit binary code
VAR_INPUT
	GreyBit0 : BOOL := FALSE ;
	GreyBit1 : BOOL := FALSE ;
	GreyBit2 : BOOL := FALSE ;
	GreyBit3 : BOOL := FALSE ;
END_VAR
VAR
	TempInt : INT ; // temporary 
END_VAR

// convert grey code into binary
TempInt.3 	:= GreyBit3 ;
TempInt.2	:= GreyBit3 	XOR GreyBit2 ;
TempInt.1	:= TempInt.2	XOR GreyBit1 ;
TempInt.0	:= TempInt.1	XOR GreyBit0 ;

Grey_To_Bin := TempInt ;

END_FUNCTION

// ---- Conversion/Rpm_To_DegS.TcPOU
(* convert rotations per minute to degrees per second *)
FUNCTION Rpm_To_DegS : LREAL 
VAR_INPUT
	Rpm : LREAL ; // input revolutions per minute
END_VAR

// ===== convert RPM to DegS ====
	Rpm_To_DegS := (Rpm/60)*360 ;

END_FUNCTION

// ---- Logger/Functions/LogHandlers/FB_LogHandler_PersistentArray.TcPOU
FUNCTION_BLOCK FB_LogHandler_PersistentArray EXTENDS FB_LogHandlerBase // Writes the last X-number of log items to a persistent list
VAR_OUTPUT PERSISTENT
	aLogItems : ARRAY[1..GVL_Utilities.RETAINABLE_LOG_HISTORY_SIZE] OF UDT_LogItem;
	nIndex : UINT; // Array index of the last added log item
END_VAR

METHOD INTERNAL FINAL AddToLog
VAR_INPUT
	stLogItem : UDT_LogItem;
END_VAR
VAR
	i : UINT; // Iterator
END_VAR
nIndex := (nIndex MOD GVL_Utilities.RETAINABLE_LOG_HISTORY_SIZE) + 1;
aLogItems[nIndex] := stLogItem;
END_METHOD

END_FUNCTION_BLOCK

// ---- Positions/Functions/F_PosCheck.TcPOU
(* Returns a true when position is within tollerance *)
FUNCTION F_PosCheck : bool
VAR_INPUT
	TargetPos		: LREAL ; // target position to check [deg]
	ActPos			: LREAL	; // Actual position [deg]
	Lowtol			: LREAL	; // Low tolerance (is reduced from target pos)
	HighTol			: LREAL	; // High tollerance (is added to target position)
	EncTurnover		: DINT 	; // Encoder turnover value
END_VAR
VAR
	Lowval	: LREAL ;
	HighVal	: LREAL ;
	LowTurn	: BOOL ;
	HighTurn: BOOL ;
	HighOk	: BOOL ;
	LowOK	: BOOL ;
END_VAR

// Check lower and uper do not exceed turnover
	IF TargetPos - Lowtol < 0 THEN 
		Lowval 	:= EncTurnover + TargetPos - Lowtol ;
		LowTurn	:= TRUE ;
	ELSE 
		LowTurn := FALSE ;
	END_IF

	IF TargetPos + HighTol > 360 THEN 
		HighVal	:= EncTurnover - TargetPos + Lowtol ;
		HighTurn:= TRUE ;
	ELSE 
		HighTurn := FALSE ;
	END_IF

	
// Check lower limit
	IF LowTurn AND ActPos > Lowval THEN
		LowOK := TRUE ; 
	ELSIF HighTurn AND ActPos < HighVal THEN 
		LowOK := TRUE ;
	ELSIF ActPos > TargetPos - Lowtol THEN
		LowOK := TRUE ;
	ELSE 
		LowOK := FALSE ;
	END_IF
	
// Check high limit
	IF HighTurn AND ActPos < HighVal THEN
		HighOk := TRUE ;
	ELSIF LowTurn AND ActPos > Lowval THEN 
		HighOk := TRUE ; 
	ELSIF ActPos < TargetPos + HighTol THEN
		HighOk := TRUE ;
	ELSE
		HighOk := FALSE ;
	END_IF
	
// Set output
	IF LowOK AND HighOk THEN
		F_PosCheck := TRUE ;
	ELSE 
		F_PosCheck := FALSE ;
	END_IF

END_FUNCTION

// ---- StepFunctions/FB_Step.TcPOU
FUNCTION_BLOCK PUBLIC FB_Step EXTENDS FB_Base
VAR_INPUT
END_VAR
VAR_OUTPUT
	nActStep	: UDINT := 0 ; // Active step
	bIdle		: BOOL	:= TRUE  ; // Stepper is idle (Step 0)
	bPaused		: BOOL 	:= FALSE ; // Stepper is paused
	bHold		: BOOL 	:= FALSE ; // Stepper is blocked for changes
	bSkipPause	: BOOL	:= FALSE ; // Pause function is skipped in this step 
	bResetting	: BOOL  := False ; // Reset is active
END_VAR
VAR
	nPreviousStep 	: UDINT ; // Previous active step
	nNextStep		: UDINT ; // Next step to activate
	nResetStep		: UDINT ; // step to which the stepper will go after reset
END_VAR

SetActiveStep();

METHOD PUBLIC CmdHold : BOOL
VAR_INPUT
END_VAR
bHold := TRUE ;

CmdHold := bHold;
END_METHOD

METHOD PUBLIC CmdNext : BOOL
VAR_INPUT
END_VAR
IF NOT bHold THEN 
	nNextStep := nActStep +	1 ;	
END_IF

CmdNext := TRUE ;
END_METHOD

METHOD PUBLIC CmdPrevious : BOOL
VAR_INPUT
END_VAR
IF NOT bHold THEN 
	nNextStep := nPreviousStep ;	
END_IF

CmdPrevious := TRUE ;
END_METHOD

METHOD PUBLIC CmdReset : BOOL
VAR_INPUT
END_VAR
bErrorActive := FALSE ;

IF nActStep <> nResetStep THEN 
	IF NOT bResetting THEN
		bResetting := TRUE ;
	ELSE
		nPreviousStep 	:= nActStep ;
		nNextStep		:= nResetStep ;
		nActStep 		:= nResetStep ;
		bResetting 		:= FALSE;
	END_IF
ELSE
	CmdReset := TRUE ; 
END_IF
END_METHOD

METHOD PUBLIC CmdToStep : BOOL
VAR_INPUT
	nStep	: UDINT ;
END_VAR
IF NOT bHold THEN 
	nNextStep := nStep ;
END_IF

CmdToStep := nNextStep = nStep ;
END_METHOD

METHOD PUBLIC Init : BOOL
VAR_INPUT
	// Location data for messages  
	nId			: UINT ; // Identification number of object
	nParentId	: UDINT ; // Id of higher level if applicable (0 = no parent)
	nResetStep	: UDINT ; // step to which the stepper wil go at reset
END_VAR
// ====== Calculate device id =====
	ExecIdentifyDevice(nId, nParentId, E_ComponentTypes.StepProgram);
	
// ===== set reset step ======
	nActStep 			:= nResetStep ;
	THIS^.nResetStep	:= nResetStep ;
END_METHOD

METHOD PRIVATE SetActiveStep : BOOL
VAR_INPUT
END_VAR
IF bResetting THEN 
	nPreviousStep 	:= nActStep ;
	nNextStep		:= nResetStep ;
	nActStep 		:= nResetStep ;
	bResetting 		:= FALSE; 
ELSIF bHold THEN 
	bHold 			:= FALSE ;
	RETURN; 
ELSIF bErrorActive THEN 
	stFault.Active			:= TRUE ;
	stFault.Description		:= 'Invalid step state';
	stFault.FaultType		:= E_FaultTypes.FF;
ELSIF NOT bCmdPause OR bSkipPause THEN 
	IF nActStep <> nNextStep THEN 
		nPreviousStep 	:=	nActStep;	
		nActStep		:= 	nNextStep;
	END_IF
END_IF

bPaused 	:= bCmdPause ;	
bSkipPause 	:= FALSE ; 
bIdle 		:= nActStep = 0 ;
END_METHOD

METHOD Public SkipPause : BOOL
VAR_INPUT
END_VAR
bSkipPause := TRUE ;

SkipPause := true ;
END_METHOD

METHOD PUBLIC StepError : BOOL
VAR_INPUT
END_VAR
bErrorActive := TRUE ;
END_METHOD

END_FUNCTION_BLOCK
